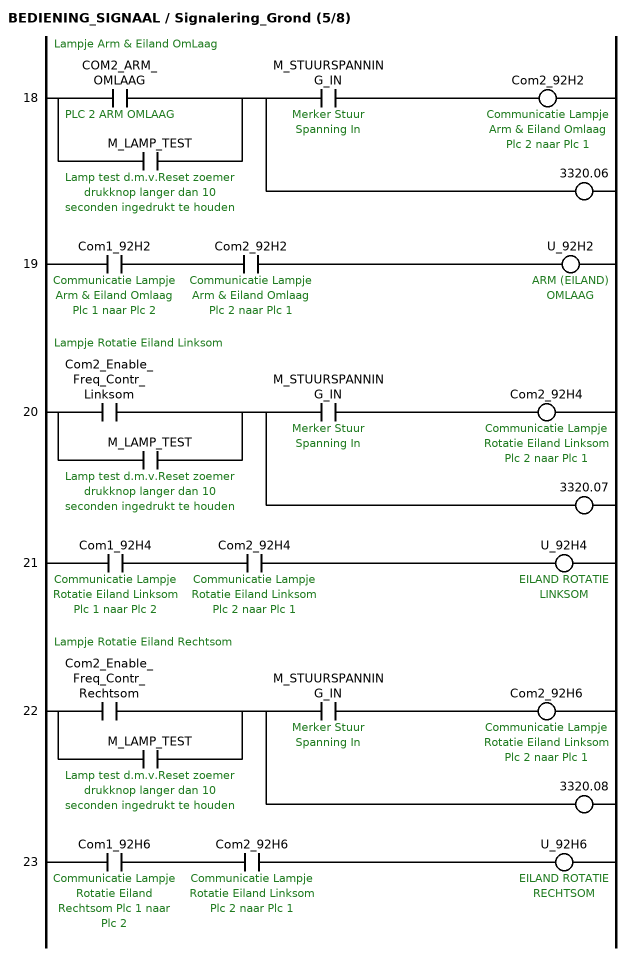
; [picture p301: BEDIENING_SIGNAAL / Signalering_Grond, rungs 18-23]
; rung 18: Lampje Arm & Eiland OmLaag
LD COM2_ARM_OMLAAG  ; PLC 2 ARM OMLAAG
OR M_LAMP_TEST  ; Lamp test d.m.v.Reset zoemer drukknop langer dan 10 seconden ingedrukt te houden
OUT TR0
AND M_STUURSPANNING_IN  ; Merker Stuur Spanning In
OUT Com2_92H2  ; Communicatie Lampje Arm & Eiland Omlaag Plc 2 naar Plc 1
LD TR0
OUT 3320.06
; rung 19
LD Com1_92H2  ; Communicatie Lampje Arm & Eiland Omlaag Plc 1 naar Plc 2
AND Com2_92H2  ; Communicatie Lampje Arm & Eiland Omlaag Plc 2 naar Plc 1
OUT U_92H2  ; ARM (EILAND) OMLAAG
; rung 20: Lampje Rotatie Eiland Linksom
LD Com2_Enable_Freq_Contr_Linksom
OR M_LAMP_TEST  ; Lamp test d.m.v.Reset zoemer drukknop langer dan 10 seconden ingedrukt te houden
OUT TR0
AND M_STUURSPANNING_IN  ; Merker Stuur Spanning In
OUT Com2_92H4  ; Communicatie Lampje Rotatie Eiland Linksom Plc 2 naar Plc 1
LD TR0
OUT 3320.07
; rung 21
LD Com1_92H4  ; Communicatie Lampje Rotatie Eiland Linksom Plc 1 naar Plc 2
AND Com2_92H4  ; Communicatie Lampje Rotatie Eiland Linksom Plc 2 naar Plc 1
OUT U_92H4  ; EILAND ROTATIE LINKSOM
; rung 22: Lampje Rotatie Eiland Rechtsom
LD Com2_Enable_Freq_Contr_Rechtsom
OR M_LAMP_TEST  ; Lamp test d.m.v.Reset zoemer drukknop langer dan 10 seconden ingedrukt te houden
OUT TR0
AND M_STUURSPANNING_IN  ; Merker Stuur Spanning In
OUT Com2_92H6  ; Communicatie Lampje Rotatie Eiland Linksom Plc 2 naar Plc 1
LD TR0
OUT 3320.08
; rung 23
LD Com1_92H6  ; Communicatie Lampje Rotatie Eiland Rechtsom Plc 1 naar Plc 2
AND Com2_92H6  ; Communicatie Lampje Rotatie Eiland Linksom Plc 2 naar Plc 1
OUT U_92H6  ; EILAND ROTATIE RECHTSOM

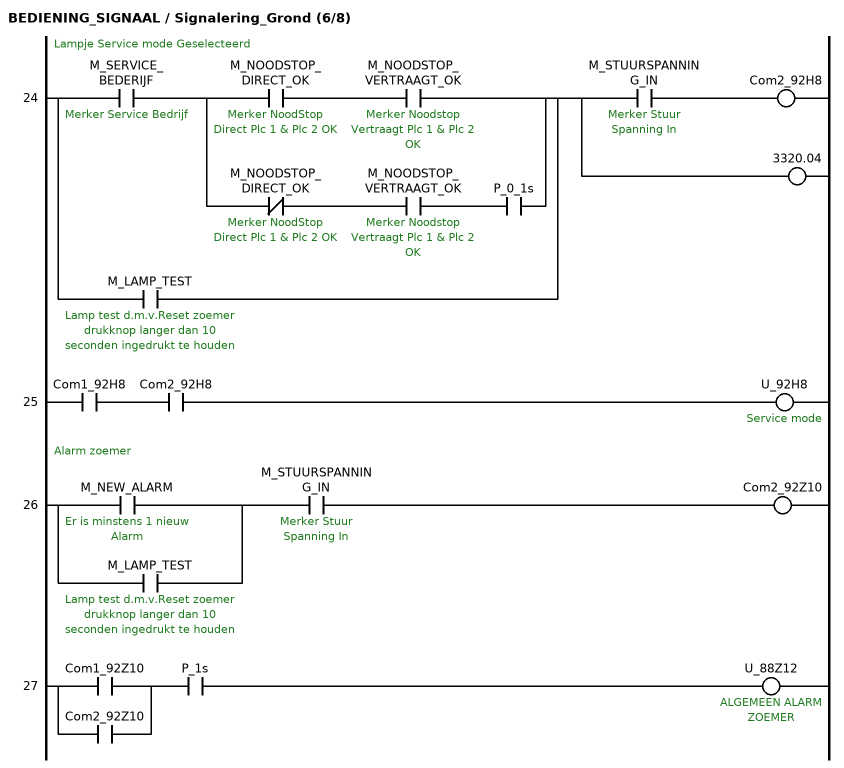
; rung 24: Lampje Service mode Geselecteerd
LD M_SERVICE_BEDERIJF  ; Merker Service Bedrijf
LD M_NOODSTOP_DIRECT_OK  ; Merker NoodStop Direct Plc 1 & Plc 2 OK
AND M_NOODSTOP_VERTRAAGT_OK  ; Merker Noodstop Vertraagt Plc 1 & Plc 2 OK
LDNOT M_NOODSTOP_DIRECT_OK  ; Merker NoodStop Direct Plc 1 & Plc 2 OK
AND M_NOODSTOP_VERTRAAGT_OK  ; Merker Noodstop Vertraagt Plc 1 & Plc 2 OK
AND P_0_1s
ORLD
ANDLD
OR M_LAMP_TEST  ; Lamp test d.m.v.Reset zoemer drukknop langer dan 10 seconden ingedrukt te houden
OUT TR0
AND M_STUURSPANNING_IN  ; Merker Stuur Spanning In
OUT Com2_92H8
LD TR0
OUT 3320.04
; rung 25
LD Com1_92H8
AND Com2_92H8
OUT U_92H8  ; Service mode
; rung 26: Alarm zoemer
LD M_NEW_ALARM  ; Er is minstens 1 nieuw Alarm
OR M_LAMP_TEST  ; Lamp test d.m.v.Reset zoemer drukknop langer dan 10 seconden ingedrukt te houden
AND M_STUURSPANNING_IN  ; Merker Stuur Spanning In
OUT Com2_92Z10
; rung 27
LD Com1_92Z10
OR Com2_92Z10
AND P_1s
OUT U_88Z12  ; ALGEMEEN ALARM ZOEMER

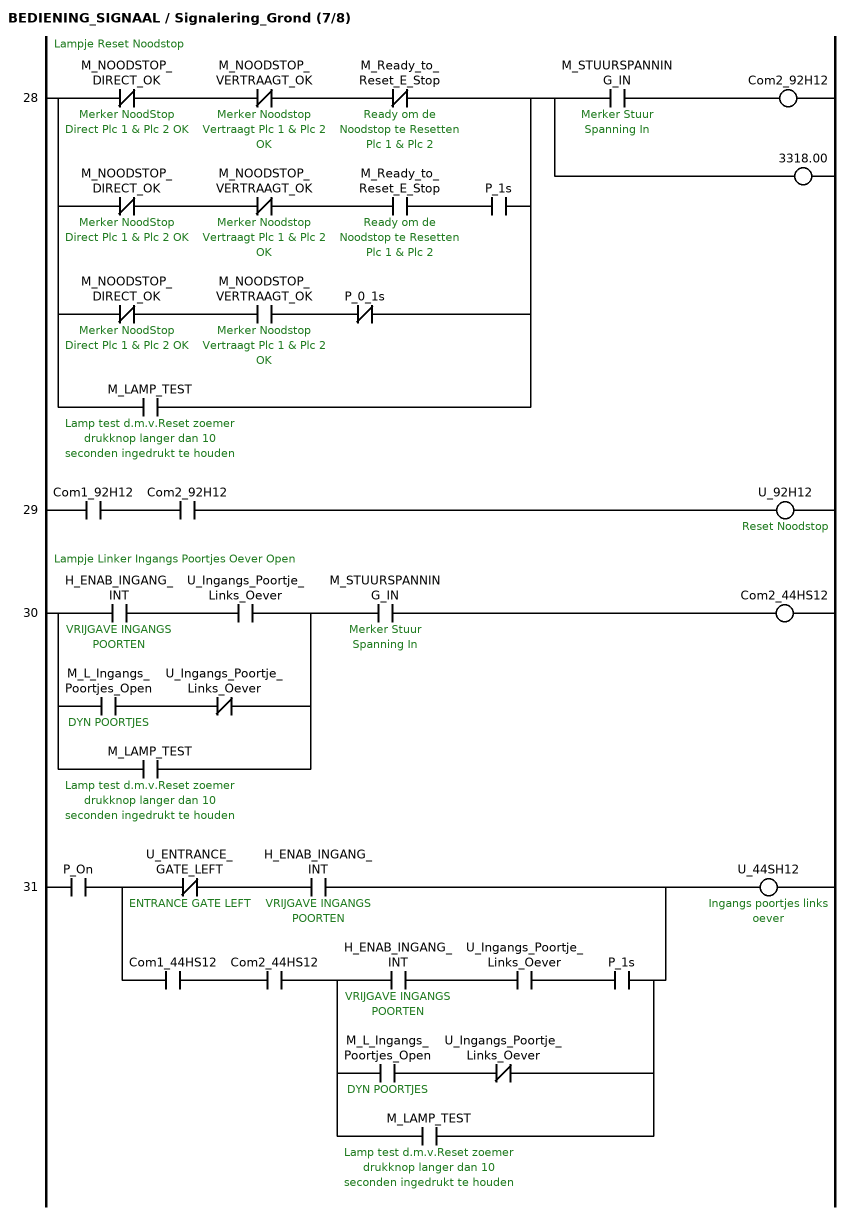
; rung 28: Lampje Reset Noodstop
LDNOT M_NOODSTOP_DIRECT_OK  ; Merker NoodStop Direct Plc 1 & Plc 2 OK
ANDNOT M_NOODSTOP_VERTRAAGT_OK  ; Merker Noodstop Vertraagt Plc 1 & Plc 2 OK
ANDNOT M_Ready_to_Reset_E_Stop  ; Ready om de Noodstop te Resetten Plc 1 & Plc 2
LDNOT M_NOODSTOP_DIRECT_OK  ; Merker NoodStop Direct Plc 1 & Plc 2 OK
ANDNOT M_NOODSTOP_VERTRAAGT_OK  ; Merker Noodstop Vertraagt Plc 1 & Plc 2 OK
AND M_Ready_to_Reset_E_Stop  ; Ready om de Noodstop te Resetten Plc 1 & Plc 2
AND P_1s
ORLD
LDNOT M_NOODSTOP_DIRECT_OK  ; Merker NoodStop Direct Plc 1 & Plc 2 OK
AND M_NOODSTOP_VERTRAAGT_OK  ; Merker Noodstop Vertraagt Plc 1 & Plc 2 OK
ANDNOT P_0_1s
ORLD
OR M_LAMP_TEST  ; Lamp test d.m.v.Reset zoemer drukknop langer dan 10 seconden ingedrukt te houden
OUT TR0
AND M_STUURSPANNING_IN  ; Merker Stuur Spanning In
OUT Com2_92H12
LD TR0
OUT 3318.00
; rung 29
LD Com1_92H12
AND Com2_92H12
OUT U_92H12  ; Reset Noodstop
; rung 30: Lampje Linker Ingangs Poortjes Oever Open
LD H_ENAB_INGANG_INT  ; VRIJGAVE INGANGS POORTEN
AND U_Ingangs_Poortje_Links_Oever
LD M_L_Ingangs_Poortjes_Open  ; DYN POORTJES
ANDNOT U_Ingangs_Poortje_Links_Oever
ORLD
OR M_LAMP_TEST  ; Lamp test d.m.v.Reset zoemer drukknop langer dan 10 seconden ingedrukt te houden
AND M_STUURSPANNING_IN  ; Merker Stuur Spanning In
OUT Com2_44HS12
; rung 31
LD P_On
LDNOT U_ENTRANCE_GATE_LEFT  ; ENTRANCE GATE LEFT
AND H_ENAB_INGANG_INT  ; VRIJGAVE INGANGS POORTEN
LD Com1_44HS12
AND Com2_44HS12
LD H_ENAB_INGANG_INT  ; VRIJGAVE INGANGS POORTEN
AND U_Ingangs_Poortje_Links_Oever
AND P_1s
LD M_L_Ingangs_Poortjes_Open  ; DYN POORTJES
ANDNOT U_Ingangs_Poortje_Links_Oever
ORLD
OR M_LAMP_TEST  ; Lamp test d.m.v.Reset zoemer drukknop langer dan 10 seconden ingedrukt te houden
ANDLD
ORLD
ANDLD
OUT U_44SH12  ; Ingangs poortjes links oever

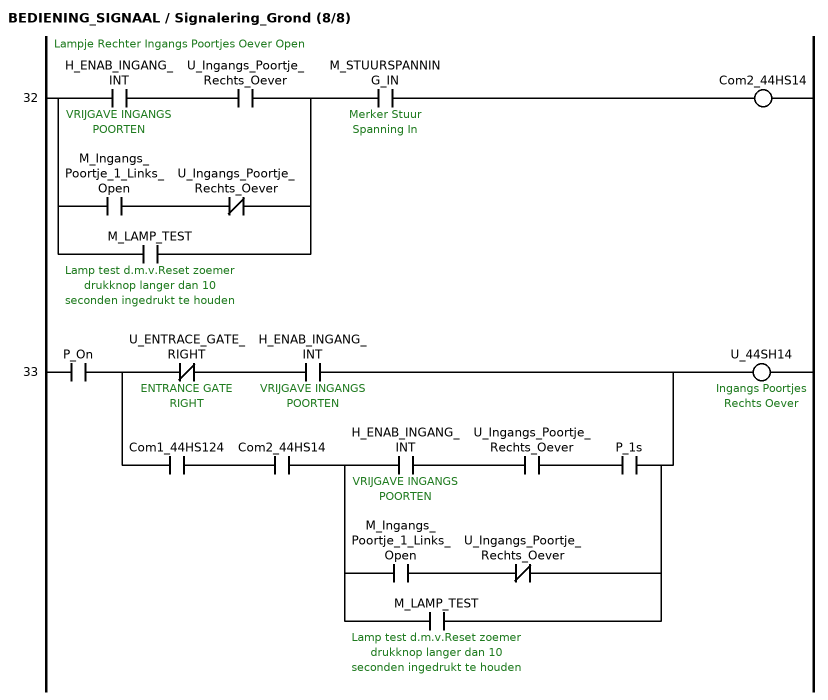
; rung 32: Lampje Rechter Ingangs Poortjes Oever Open
LD H_ENAB_INGANG_INT  ; VRIJGAVE INGANGS POORTEN
AND U_Ingangs_Poortje_Rechts_Oever
LD M_Ingangs_Poortje_1_Links_Open
ANDNOT U_Ingangs_Poortje_Rechts_Oever
ORLD
OR M_LAMP_TEST  ; Lamp test d.m.v.Reset zoemer drukknop langer dan 10 seconden ingedrukt te houden
AND M_STUURSPANNING_IN  ; Merker Stuur Spanning In
OUT Com2_44HS14
; rung 33
LD P_On
LDNOT U_ENTRACE_GATE_RIGHT  ; ENTRANCE GATE RIGHT
AND H_ENAB_INGANG_INT  ; VRIJGAVE INGANGS POORTEN
LD Com1_44HS124
AND Com2_44HS14
LD H_ENAB_INGANG_INT  ; VRIJGAVE INGANGS POORTEN
AND U_Ingangs_Poortje_Rechts_Oever
AND P_1s
LD M_Ingangs_Poortje_1_Links_Open
ANDNOT U_Ingangs_Poortje_Rechts_Oever
ORLD
OR M_LAMP_TEST  ; Lamp test d.m.v.Reset zoemer drukknop langer dan 10 seconden ingedrukt te houden
ANDLD
ORLD
ANDLD
OUT U_44SH14  ; Ingangs Poortjes Rechts Oever

### Section Bediening_Eiland

### Section Signalering_Eiland

### Section Bediening_Display_Eiland

### Section Signalering_Display_Eiland

### Section Einde_Bediening_Signalering
; rung 0
END(001)

## Program HOOFD_BESTURING (cyclic task 2)

### Section Automatische_Afloop_In_Uitgangs_Poortjes

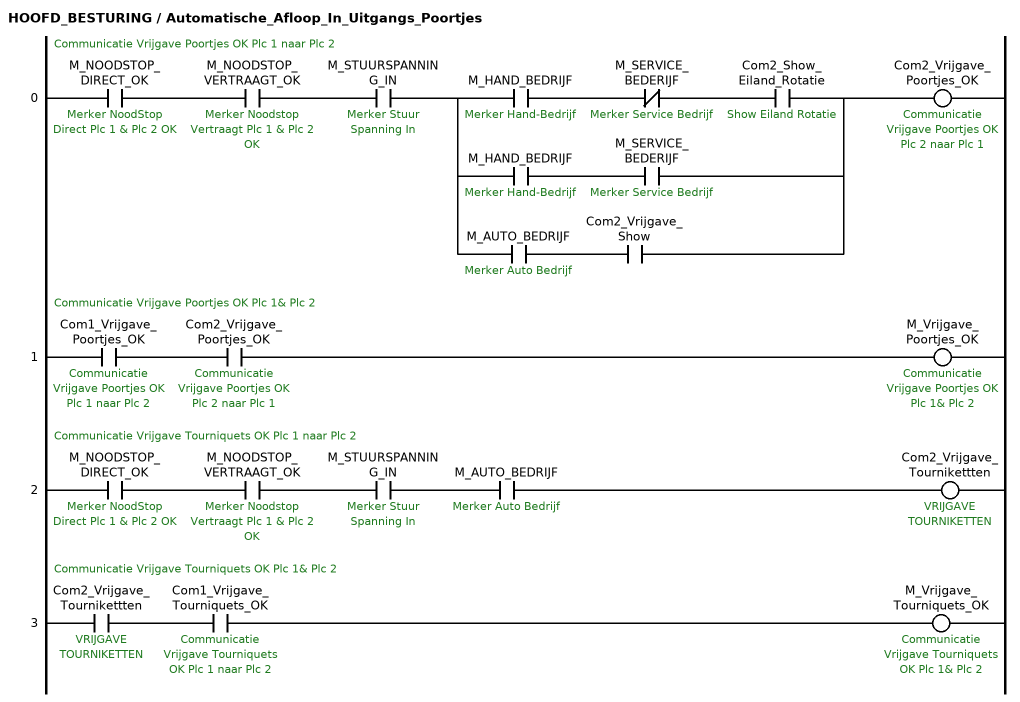
; rung 0: Communicatie Vrijgave Poortjes OK Plc 1 naar Plc 2
LD M_NOODSTOP_DIRECT_OK  ; Merker NoodStop Direct Plc 1 & Plc 2 OK
AND M_NOODSTOP_VERTRAAGT_OK  ; Merker Noodstop Vertraagt Plc 1 & Plc 2 OK
AND M_STUURSPANNING_IN  ; Merker Stuur Spanning In
LD M_HAND_BEDRIJF  ; Merker Hand-Bedrijf
ANDNOT M_SERVICE_BEDERIJF  ; Merker Service Bedrijf
AND Com2_Show_Eiland_Rotatie  ; Show Eiland Rotatie
LD M_HAND_BEDRIJF  ; Merker Hand-Bedrijf
AND M_SERVICE_BEDERIJF  ; Merker Service Bedrijf
ORLD
LD M_AUTO_BEDRIJF  ; Merker Auto Bedrijf
AND Com2_Vrijgave_Show
ORLD
ANDLD
OUT Com2_Vrijgave_Poortjes_OK  ; Communicatie Vrijgave Poortjes OK Plc 2 naar Plc 1
; rung 1: Communicatie Vrijgave Poortjes OK Plc 1& Plc 2
LD Com1_Vrijgave_Poortjes_OK  ; Communicatie Vrijgave Poortjes OK Plc 1 naar Plc 2
AND Com2_Vrijgave_Poortjes_OK  ; Communicatie Vrijgave Poortjes OK Plc 2 naar Plc 1
OUT M_Vrijgave_Poortjes_OK  ; Communicatie Vrijgave Poortjes OK Plc 1& Plc 2
; rung 2: Communicatie Vrijgave Tourniquets OK Plc 1 naar Plc 2
LD M_NOODSTOP_DIRECT_OK  ; Merker NoodStop Direct Plc 1 & Plc 2 OK
AND M_NOODSTOP_VERTRAAGT_OK  ; Merker Noodstop Vertraagt Plc 1 & Plc 2 OK
AND M_STUURSPANNING_IN  ; Merker Stuur Spanning In
AND M_AUTO_BEDRIJF  ; Merker Auto Bedrijf
OUT Com2_Vrijgave_Tournikettten  ; VRIJGAVE TOURNIKETTEN
; rung 3: Communicatie Vrijgave Tourniquets OK Plc 1& Plc 2
LD Com2_Vrijgave_Tournikettten  ; VRIJGAVE TOURNIKETTEN
AND Com1_Vrijgave_Tourniquets_OK  ; Communicatie Vrijgave Tourniquets OK Plc 1 naar Plc 2
OUT M_Vrijgave_Tourniquets_OK  ; Communicatie Vrijgave Tourniquets OK Plc 1& Plc 2

### Section Automatisch_Programma_Afloop

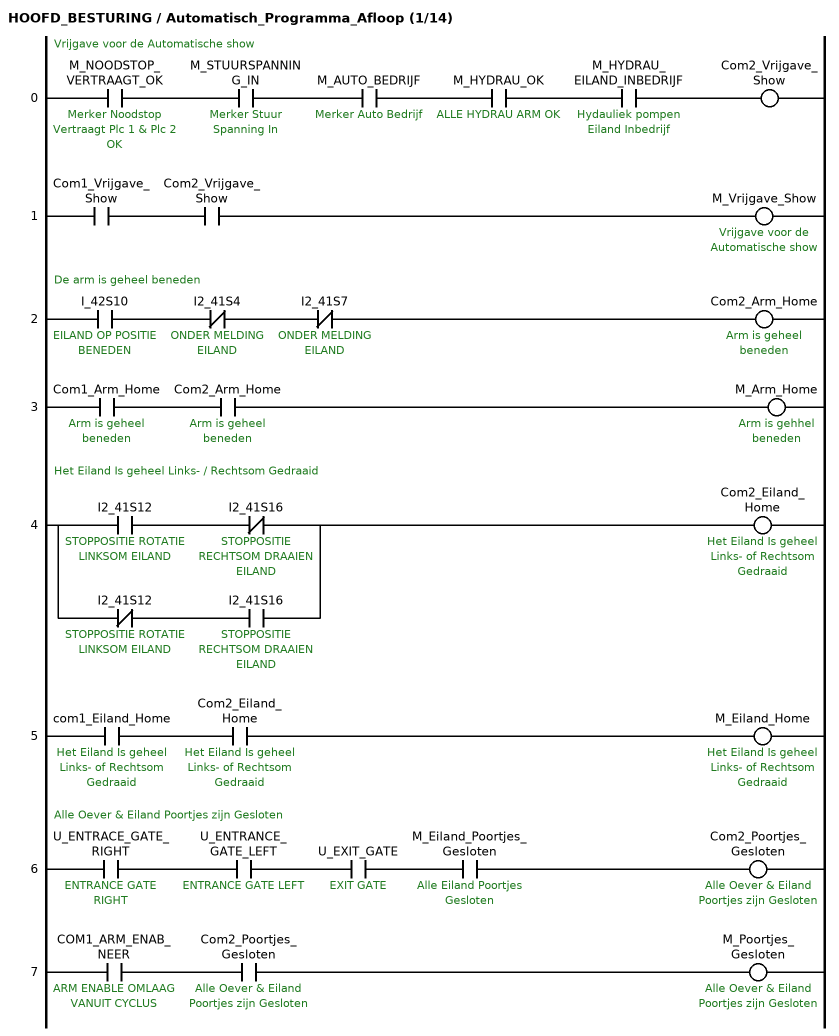
; rung 0: Vrijgave voor de Automatische show
LD M_NOODSTOP_VERTRAAGT_OK  ; Merker Noodstop Vertraagt Plc 1 & Plc 2 OK
AND M_STUURSPANNING_IN  ; Merker Stuur Spanning In
AND M_AUTO_BEDRIJF  ; Merker Auto Bedrijf
AND M_HYDRAU_OK  ; ALLE HYDRAU ARM OK
AND M_HYDRAU_EILAND_INBEDRIJF  ; Hydauliek pompen Eiland Inbedrijf
OUT Com2_Vrijgave_Show
; rung 1
LD Com1_Vrijgave_Show
AND Com2_Vrijgave_Show
OUT M_Vrijgave_Show  ; Vrijgave voor de Automatische show
; rung 2: De arm is geheel beneden
LD I_42S10  ; EILAND OP POSITIE BENEDEN
ANDNOT I2_41S4  ; ONDER MELDING EILAND
ANDNOT I2_41S7  ; ONDER MELDING EILAND
OUT Com2_Arm_Home  ; Arm is geheel beneden
; rung 3
LD Com1_Arm_Home  ; Arm is geheel beneden
AND Com2_Arm_Home  ; Arm is geheel beneden
OUT M_Arm_Home  ; Arm is gehhel beneden
; rung 4: Het Eiland Is geheel Links- / Rechtsom Gedraaid
LD I2_41S12  ; STOPPOSITIE ROTATIE LINKSOM EILAND
ANDNOT I2_41S16  ; STOPPOSITIE RECHTSOM DRAAIEN EILAND
LDNOT I2_41S12  ; STOPPOSITIE ROTATIE LINKSOM EILAND
AND I2_41S16  ; STOPPOSITIE RECHTSOM DRAAIEN EILAND
ORLD
OUT Com2_Eiland_Home  ; Het Eiland Is geheel Links- of Rechtsom Gedraaid
; rung 5
LD com1_Eiland_Home  ; Het Eiland Is geheel Links- of Rechtsom Gedraaid
AND Com2_Eiland_Home  ; Het Eiland Is geheel Links- of Rechtsom Gedraaid
OUT M_Eiland_Home  ; Het Eiland Is geheel Links- of Rechtsom Gedraaid
; rung 6: Alle Oever & Eiland Poortjes zijn Gesloten
LD U_ENTRACE_GATE_RIGHT  ; ENTRANCE GATE RIGHT
AND U_ENTRANCE_GATE_LEFT  ; ENTRANCE GATE LEFT
AND U_EXIT_GATE  ; EXIT GATE
AND M_Eiland_Poortjes_Gesloten  ; Alle Eiland Poortjes Gesloten
OUT Com2_Poortjes_Gesloten  ; Alle Oever & Eiland Poortjes zijn Gesloten
; rung 7
LD COM1_ARM_ENAB_NEER  ; ARM ENABLE OMLAAG  VANUIT CYCLUS
AND Com2_Poortjes_Gesloten  ; Alle Oever & Eiland Poortjes zijn Gesloten
OUT M_Poortjes_Gesloten  ; Alle Oever & Eiland Poortjes zijn Gesloten

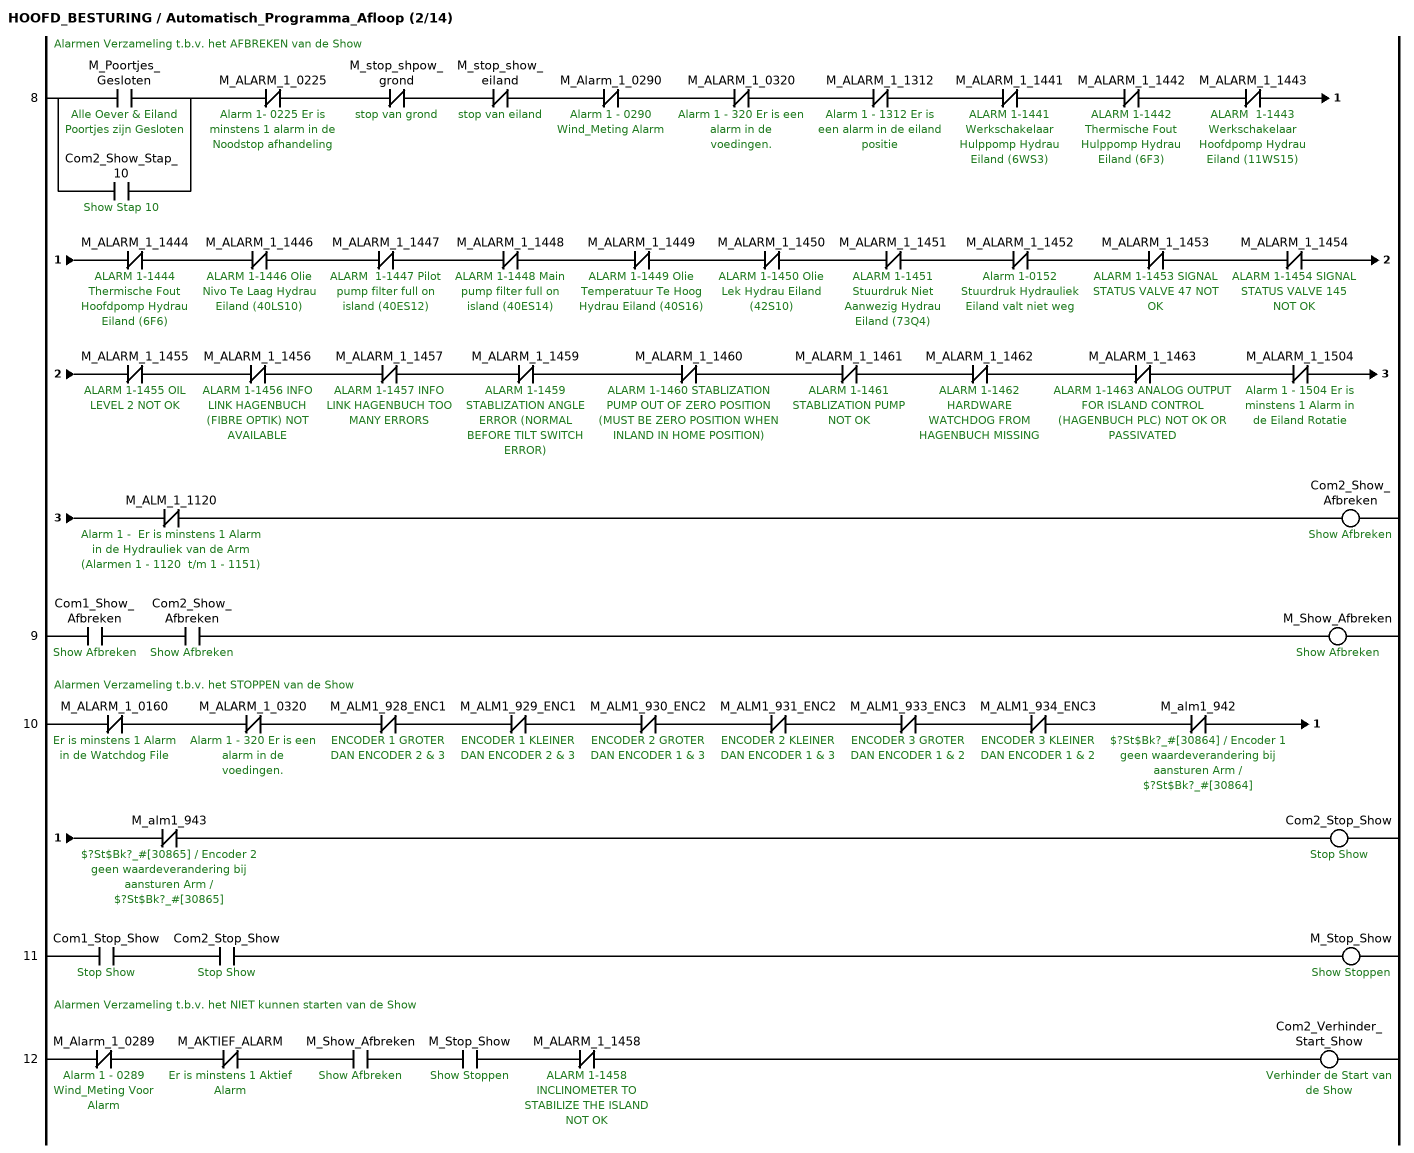
; rung 8: Alarmen Verzameling t.b.v. het AFBREKEN van de Show
LD M_Poortjes_Gesloten  ; Alle Oever & Eiland Poortjes zijn Gesloten
OR Com2_Show_Stap_10  ; Show Stap 10
ANDNOT M_ALARM_1_0225  ; Alarm 1- 0225 Er is minstens 1 alarm in de Noodstop afhandeling
ANDNOT M_stop_shpow_grond  ; stop van grond
ANDNOT M_stop_show_eiland  ; stop van eiland
ANDNOT M_Alarm_1_0290  ; Alarm 1 - 0290 Wind_Meting Alarm
ANDNOT M_ALARM_1_0320  ; Alarm 1 - 320 Er is een alarm in de voedingen.
ANDNOT M_ALARM_1_1312  ; Alarm 1 - 1312 Er is een alarm in de eiland positie
ANDNOT M_ALARM_1_1441  ; ALARM 1-1441 Werkschakelaar Hulppomp Hydrau Eiland (6WS3)
ANDNOT M_ALARM_1_1442  ; ALARM 1-1442 Thermische Fout Hulppomp Hydrau Eiland (6F3)
ANDNOT M_ALARM_1_1443  ; ALARM  1-1443 Werkschakelaar Hoofdpomp Hydrau Eiland (11WS15)
ANDNOT M_ALARM_1_1444  ; ALARM 1-1444 Thermische Fout Hoofdpomp Hydrau Eiland (6F6)
ANDNOT M_ALARM_1_1446  ; ALARM 1-1446 Olie Nivo Te Laag Hydrau Eiland (40LS10)
ANDNOT M_ALARM_1_1447  ; ALARM  1-1447 Pilot pump filter full on island (40ES12)
ANDNOT M_ALARM_1_1448  ; ALARM 1-1448 Main pump filter full on island (40ES14)
ANDNOT M_ALARM_1_1449  ; ALARM 1-1449 Olie Temperatuur Te Hoog Hydrau Eiland (40S16)
ANDNOT M_ALARM_1_1450  ; ALARM 1-1450 Olie Lek Hydrau Eiland (42S10)
ANDNOT M_ALARM_1_1451  ; ALARM 1-1451 Stuurdruk Niet Aanwezig Hydrau Eiland (73Q4)
ANDNOT M_ALARM_1_1452  ; Alarm 1-0152 Stuurdruk Hydrauliek Eiland valt niet weg
ANDNOT M_ALARM_1_1453  ; ALARM 1-1453 SIGNAL STATUS VALVE 47 NOT OK
ANDNOT M_ALARM_1_1454  ; ALARM 1-1454 SIGNAL STATUS VALVE 145 NOT OK
ANDNOT M_ALARM_1_1455  ; ALARM 1-1455 OIL LEVEL 2 NOT OK
ANDNOT M_ALARM_1_1456  ; ALARM 1-1456 INFO LINK HAGENBUCH (FIBRE OPTIK) NOT AVAILABLE
ANDNOT M_ALARM_1_1457  ; ALARM 1-1457 INFO LINK HAGENBUCH TOO MANY ERRORS
ANDNOT M_ALARM_1_1459  ; ALARM 1-1459 STABLIZATION ANGLE ERROR (NORMAL BEFORE TILT SWITCH ERROR)
ANDNOT M_ALARM_1_1460  ; ALARM 1-1460 STABLIZATION PUMP OUT OF ZERO POSITION (MUST BE ZERO POSITION WHEN INLAND IN HOME POSITION)
ANDNOT M_ALARM_1_1461  ; ALARM 1-1461 STABLIZATION PUMP NOT OK
ANDNOT M_ALARM_1_1462  ; ALARM 1-1462 HARDWARE WATCHDOG FROM HAGENBUCH MISSING
ANDNOT M_ALARM_1_1463  ; ALARM 1-1463 ANALOG OUTPUT FOR ISLAND CONTROL (HAGENBUCH PLC) NOT OK OR PASSIVATED
ANDNOT M_ALARM_1_1504  ; Alarm 1 - 1504 Er is minstens 1 Alarm in de Eiland Rotatie
ANDNOT M_ALM_1_1120  ; Alarm 1 -  Er is minstens 1 Alarm in de Hydrauliek van de Arm  (Alarmen 1 - 1120  t/m 1 - 1151)
OUT Com2_Show_Afbreken  ; Show Afbreken
; rung 9
LD Com1_Show_Afbreken  ; Show Afbreken
AND Com2_Show_Afbreken  ; Show Afbreken
OUT M_Show_Afbreken  ; Show Afbreken
; rung 10: Alarmen Verzameling t.b.v. het STOPPEN van de Show
LDNOT M_ALARM_1_0160  ; Er is minstens 1 Alarm in de Watchdog File
ANDNOT M_ALARM_1_0320  ; Alarm 1 - 320 Er is een alarm in de voedingen.
ANDNOT M_ALM1_928_ENC1  ; ENCODER 1 GROTER DAN ENCODER 2 & 3
ANDNOT M_ALM1_929_ENC1  ; ENCODER 1 KLEINER DAN ENCODER 2 & 3
ANDNOT M_ALM1_930_ENC2  ; ENCODER 2 GROTER DAN ENCODER 1 & 3
ANDNOT M_ALM1_931_ENC2  ; ENCODER 2 KLEINER DAN ENCODER 1 & 3
ANDNOT M_ALM1_933_ENC3  ; ENCODER 3 GROTER DAN ENCODER 1 & 2
ANDNOT M_ALM1_934_ENC3  ; ENCODER 3 KLEINER DAN ENCODER 1 & 2
ANDNOT M_alm1_942  ; $?St$Bk?_#[30864] / Encoder 1 geen waardeverandering bij aansturen Arm / $?St$Bk?_#[30864]
ANDNOT M_alm1_943  ; $?St$Bk?_#[30865] / Encoder 2 geen waardeverandering bij aansturen Arm / $?St$Bk?_#[30865]
OUT Com2_Stop_Show  ; Stop Show
; rung 11
LD Com1_Stop_Show  ; Stop Show
AND Com2_Stop_Show  ; Stop Show
OUT M_Stop_Show  ; Show Stoppen
; rung 12: Alarmen Verzameling t.b.v. het NIET kunnen starten van de Show
LDNOT M_Alarm_1_0289  ; Alarm 1 - 0289 Wind_Meting Voor Alarm
ANDNOT M_AKTIEF_ALARM  ; Er is minstens 1 Aktief Alarm
AND M_Show_Afbreken  ; Show Afbreken
AND M_Stop_Show  ; Show Stoppen
ANDNOT M_ALARM_1_1458  ; ALARM 1-1458 INCLINOMETER TO STABILIZE THE ISLAND NOT OK
OUT Com2_Verhinder_Start_Show  ; Verhinder de Start van de Show

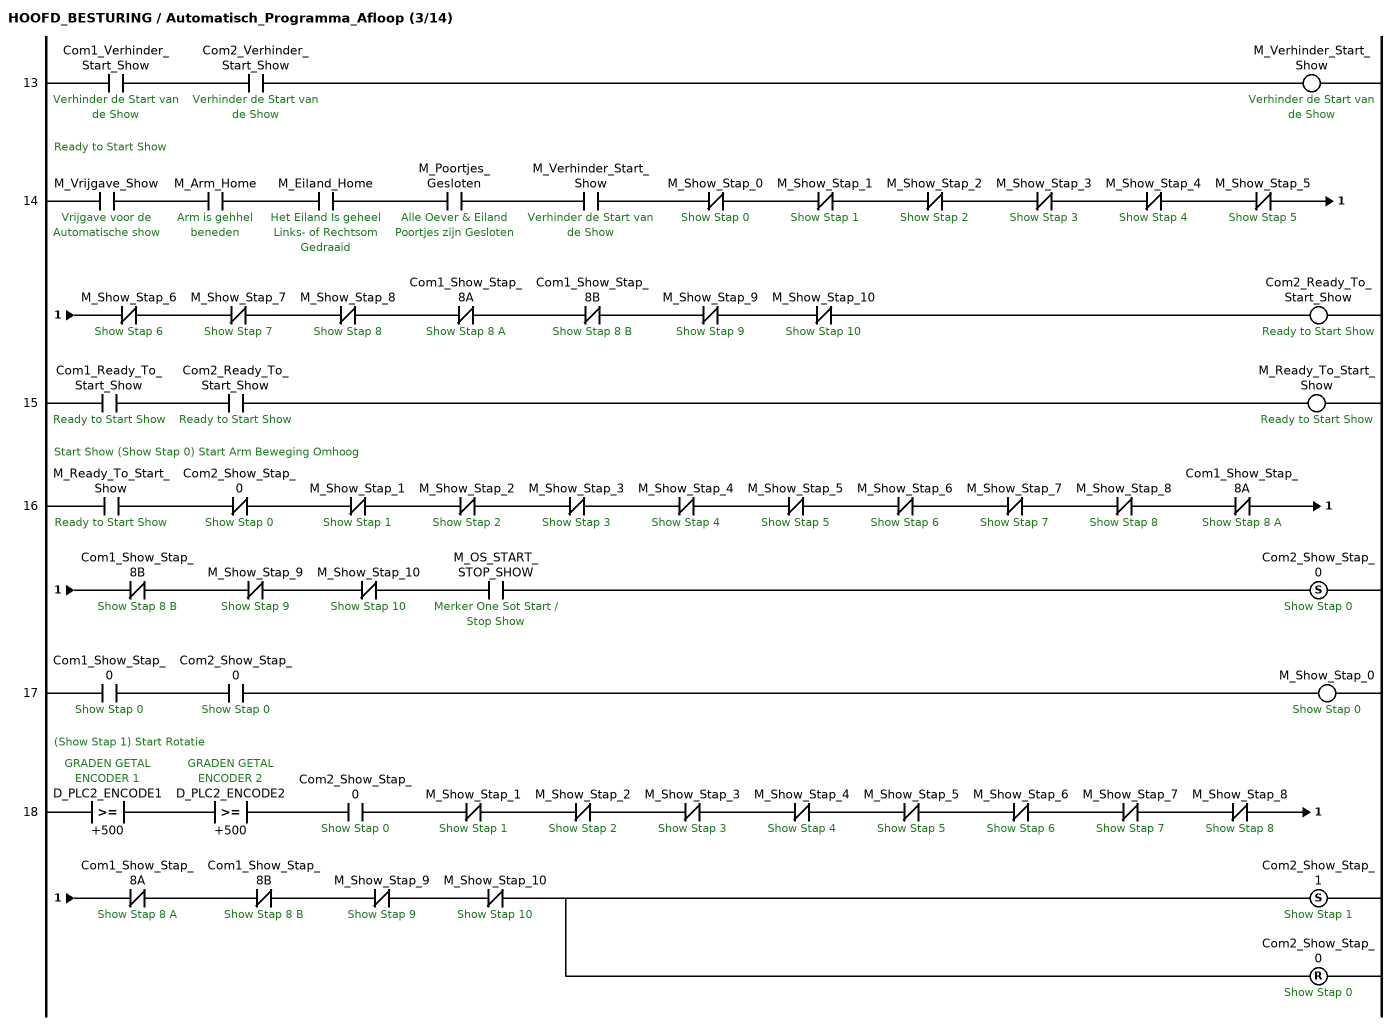
; rung 13
LD Com1_Verhinder_Start_Show  ; Verhinder de Start van de Show
AND Com2_Verhinder_Start_Show  ; Verhinder de Start van de Show
OUT M_Verhinder_Start_Show  ; Verhinder de Start van de Show
; rung 14: Ready to Start Show
LD M_Vrijgave_Show  ; Vrijgave voor de Automatische show
AND M_Arm_Home  ; Arm is gehhel beneden
AND M_Eiland_Home  ; Het Eiland Is geheel Links- of Rechtsom Gedraaid
AND M_Poortjes_Gesloten  ; Alle Oever & Eiland Poortjes zijn Gesloten
AND M_Verhinder_Start_Show  ; Verhinder de Start van de Show
ANDNOT M_Show_Stap_0  ; Show Stap 0
ANDNOT M_Show_Stap_1  ; Show Stap 1
ANDNOT M_Show_Stap_2  ; Show Stap 2
ANDNOT M_Show_Stap_3  ; Show Stap 3
ANDNOT M_Show_Stap_4  ; Show Stap 4
ANDNOT M_Show_Stap_5  ; Show Stap 5
ANDNOT M_Show_Stap_6  ; Show Stap 6
ANDNOT M_Show_Stap_7  ; Show Stap 7
ANDNOT M_Show_Stap_8  ; Show Stap 8
ANDNOT Com1_Show_Stap_8A  ; Show Stap 8 A
ANDNOT Com1_Show_Stap_8B  ; Show Stap 8 B
ANDNOT M_Show_Stap_9  ; Show Stap 9
ANDNOT M_Show_Stap_10  ; Show Stap 10
OUT Com2_Ready_To_Start_Show  ; Ready to Start Show
; rung 15
LD Com1_Ready_To_Start_Show  ; Ready to Start Show
AND Com2_Ready_To_Start_Show  ; Ready to Start Show
OUT M_Ready_To_Start_Show  ; Ready to Start Show
; rung 16: Start Show (Show Stap 0) Start Arm Beweging Omhoog
LD M_Ready_To_Start_Show  ; Ready to Start Show
ANDNOT Com2_Show_Stap_0  ; Show Stap 0
ANDNOT M_Show_Stap_1  ; Show Stap 1
ANDNOT M_Show_Stap_2  ; Show Stap 2
ANDNOT M_Show_Stap_3  ; Show Stap 3
ANDNOT M_Show_Stap_4  ; Show Stap 4
ANDNOT M_Show_Stap_5  ; Show Stap 5
ANDNOT M_Show_Stap_6  ; Show Stap 6
ANDNOT M_Show_Stap_7  ; Show Stap 7
ANDNOT M_Show_Stap_8  ; Show Stap 8
ANDNOT Com1_Show_Stap_8A  ; Show Stap 8 A
ANDNOT Com1_Show_Stap_8B  ; Show Stap 8 B
ANDNOT M_Show_Stap_9  ; Show Stap 9
ANDNOT M_Show_Stap_10  ; Show Stap 10
AND M_OS_START_STOP_SHOW  ; Merker One Sot Start / Stop Show
SET Com2_Show_Stap_0  ; Show Stap 0
; rung 17
LD Com1_Show_Stap_0  ; Show Stap 0
AND Com2_Show_Stap_0  ; Show Stap 0
OUT M_Show_Stap_0  ; Show Stap 0
; rung 18: (Show Stap 1) Start Rotatie
LD>=S(327) D_PLC2_ENCODE1 +500  ; GRADEN GETAL ENCODER 1
AND>=S(327) D_PLC2_ENCODE2 +500  ; GRADEN GETAL ENCODER 2
AND Com2_Show_Stap_0  ; Show Stap 0
ANDNOT M_Show_Stap_1  ; Show Stap 1
ANDNOT M_Show_Stap_2  ; Show Stap 2
ANDNOT M_Show_Stap_3  ; Show Stap 3
ANDNOT M_Show_Stap_4  ; Show Stap 4
ANDNOT M_Show_Stap_5  ; Show Stap 5
ANDNOT M_Show_Stap_6  ; Show Stap 6
ANDNOT M_Show_Stap_7  ; Show Stap 7
ANDNOT M_Show_Stap_8  ; Show Stap 8
ANDNOT Com1_Show_Stap_8A  ; Show Stap 8 A
ANDNOT Com1_Show_Stap_8B  ; Show Stap 8 B
ANDNOT M_Show_Stap_9  ; Show Stap 9
ANDNOT M_Show_Stap_10  ; Show Stap 10
SET Com2_Show_Stap_1  ; Show Stap 1
RSET Com2_Show_Stap_0  ; Show Stap 0

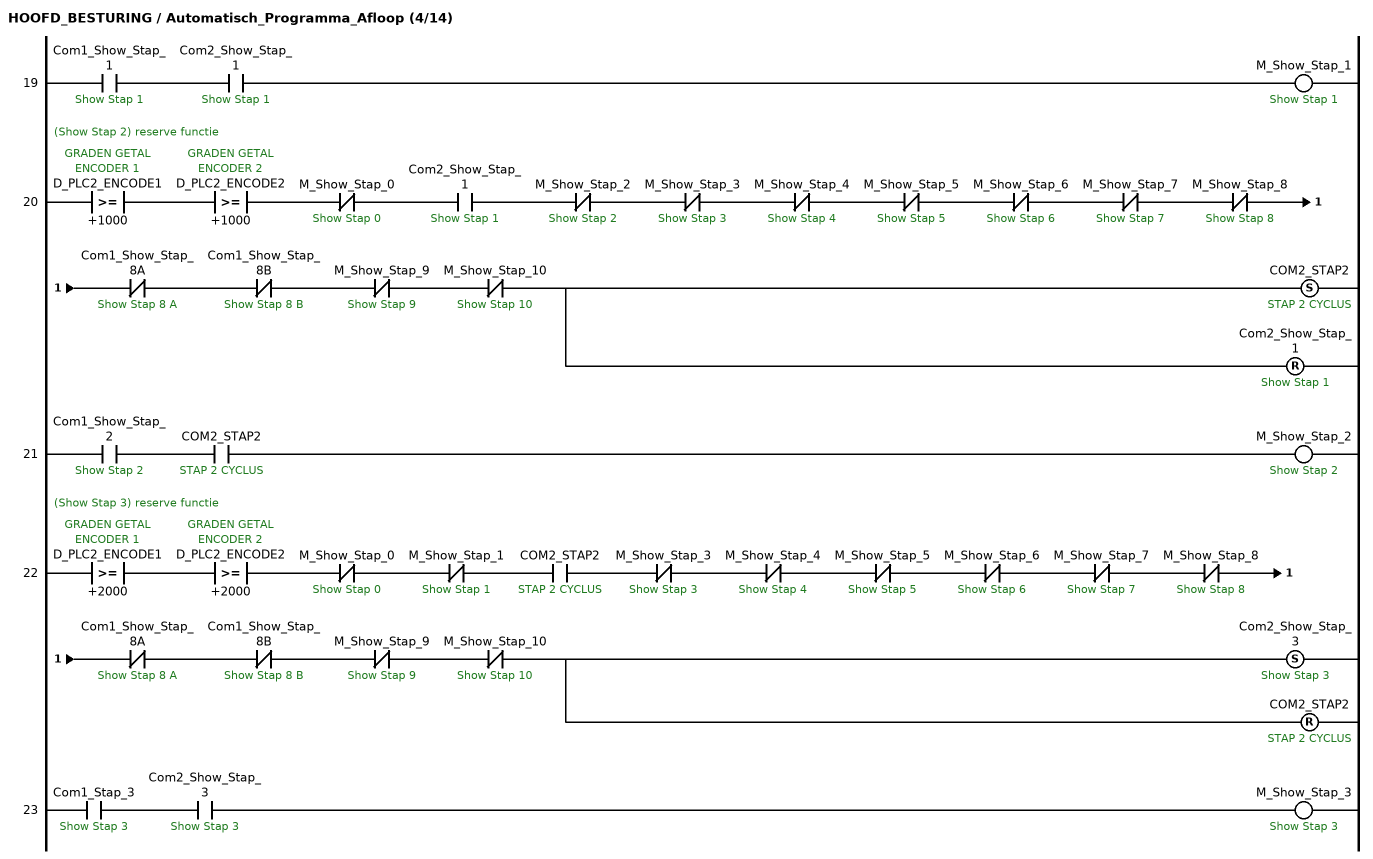
; rung 19
LD Com1_Show_Stap_1  ; Show Stap 1
AND Com2_Show_Stap_1  ; Show Stap 1
OUT M_Show_Stap_1  ; Show Stap 1
; rung 20: (Show Stap 2) reserve functie
LD>=S(327) D_PLC2_ENCODE1 +1000  ; GRADEN GETAL ENCODER 1
AND>=S(327) D_PLC2_ENCODE2 +1000  ; GRADEN GETAL ENCODER 2
ANDNOT M_Show_Stap_0  ; Show Stap 0
AND Com2_Show_Stap_1  ; Show Stap 1
ANDNOT M_Show_Stap_2  ; Show Stap 2
ANDNOT M_Show_Stap_3  ; Show Stap 3
ANDNOT M_Show_Stap_4  ; Show Stap 4
ANDNOT M_Show_Stap_5  ; Show Stap 5
ANDNOT M_Show_Stap_6  ; Show Stap 6
ANDNOT M_Show_Stap_7  ; Show Stap 7
ANDNOT M_Show_Stap_8  ; Show Stap 8
ANDNOT Com1_Show_Stap_8A  ; Show Stap 8 A
ANDNOT Com1_Show_Stap_8B  ; Show Stap 8 B
ANDNOT M_Show_Stap_9  ; Show Stap 9
ANDNOT M_Show_Stap_10  ; Show Stap 10
SET COM2_STAP2  ; STAP 2 CYCLUS
RSET Com2_Show_Stap_1  ; Show Stap 1
; rung 21
LD Com1_Show_Stap_2  ; Show Stap 2
AND COM2_STAP2  ; STAP 2 CYCLUS
OUT M_Show_Stap_2  ; Show Stap 2
; rung 22: (Show Stap 3) reserve functie
LD>=S(327) D_PLC2_ENCODE1 +2000  ; GRADEN GETAL ENCODER 1
AND>=S(327) D_PLC2_ENCODE2 +2000  ; GRADEN GETAL ENCODER 2
ANDNOT M_Show_Stap_0  ; Show Stap 0
ANDNOT M_Show_Stap_1  ; Show Stap 1
AND COM2_STAP2  ; STAP 2 CYCLUS
ANDNOT M_Show_Stap_3  ; Show Stap 3
ANDNOT M_Show_Stap_4  ; Show Stap 4
ANDNOT M_Show_Stap_5  ; Show Stap 5
ANDNOT M_Show_Stap_6  ; Show Stap 6
ANDNOT M_Show_Stap_7  ; Show Stap 7
ANDNOT M_Show_Stap_8  ; Show Stap 8
ANDNOT Com1_Show_Stap_8A  ; Show Stap 8 A
ANDNOT Com1_Show_Stap_8B  ; Show Stap 8 B
ANDNOT M_Show_Stap_9  ; Show Stap 9
ANDNOT M_Show_Stap_10  ; Show Stap 10
SET Com2_Show_Stap_3  ; Show Stap 3
RSET COM2_STAP2  ; STAP 2 CYCLUS
; rung 23
LD Com1_Stap_3  ; Show Stap 3
AND Com2_Show_Stap_3  ; Show Stap 3
OUT M_Show_Stap_3  ; Show Stap 3

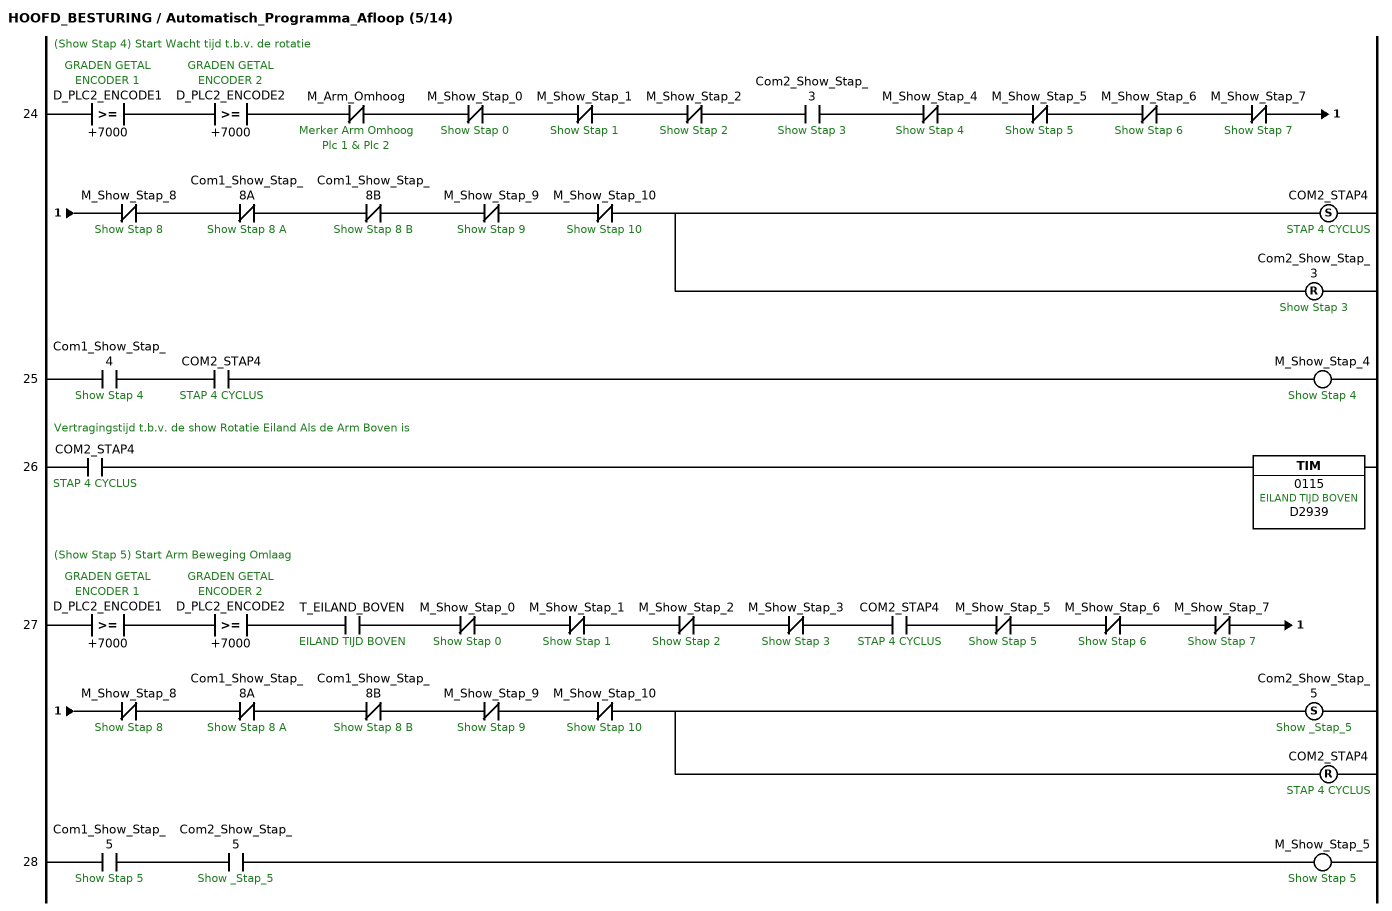
; rung 24: (Show Stap 4) Start Wacht tijd t.b.v. de rotatie
LD>=S(327) D_PLC2_ENCODE1 +7000  ; GRADEN GETAL ENCODER 1
AND>=S(327) D_PLC2_ENCODE2 +7000  ; GRADEN GETAL ENCODER 2
ANDNOT M_Arm_Omhoog  ; Merker Arm Omhoog Plc 1 & Plc 2
ANDNOT M_Show_Stap_0  ; Show Stap 0
ANDNOT M_Show_Stap_1  ; Show Stap 1
ANDNOT M_Show_Stap_2  ; Show Stap 2
AND Com2_Show_Stap_3  ; Show Stap 3
ANDNOT M_Show_Stap_4  ; Show Stap 4
ANDNOT M_Show_Stap_5  ; Show Stap 5
ANDNOT M_Show_Stap_6  ; Show Stap 6
ANDNOT M_Show_Stap_7  ; Show Stap 7
ANDNOT M_Show_Stap_8  ; Show Stap 8
ANDNOT Com1_Show_Stap_8A  ; Show Stap 8 A
ANDNOT Com1_Show_Stap_8B  ; Show Stap 8 B
ANDNOT M_Show_Stap_9  ; Show Stap 9
ANDNOT M_Show_Stap_10  ; Show Stap 10
SET COM2_STAP4  ; STAP 4 CYCLUS
RSET Com2_Show_Stap_3  ; Show Stap 3
; rung 25
LD Com1_Show_Stap_4  ; Show Stap 4
AND COM2_STAP4  ; STAP 4 CYCLUS
OUT M_Show_Stap_4  ; Show Stap 4
; rung 26: Vertragingstijd t.b.v. de show Rotatie Eiland Als de Arm Boven is
LD COM2_STAP4  ; STAP 4 CYCLUS
TIM 0115 D2939  ; EILAND TIJD BOVEN
; rung 27: (Show Stap 5) Start Arm Beweging Omlaag
LD>=S(327) D_PLC2_ENCODE1 +7000  ; GRADEN GETAL ENCODER 1
AND>=S(327) D_PLC2_ENCODE2 +7000  ; GRADEN GETAL ENCODER 2
AND T_EILAND_BOVEN  ; EILAND TIJD BOVEN
ANDNOT M_Show_Stap_0  ; Show Stap 0
ANDNOT M_Show_Stap_1  ; Show Stap 1
ANDNOT M_Show_Stap_2  ; Show Stap 2
ANDNOT M_Show_Stap_3  ; Show Stap 3
AND COM2_STAP4  ; STAP 4 CYCLUS
ANDNOT M_Show_Stap_5  ; Show Stap 5
ANDNOT M_Show_Stap_6  ; Show Stap 6
ANDNOT M_Show_Stap_7  ; Show Stap 7
ANDNOT M_Show_Stap_8  ; Show Stap 8
ANDNOT Com1_Show_Stap_8A  ; Show Stap 8 A
ANDNOT Com1_Show_Stap_8B  ; Show Stap 8 B
ANDNOT M_Show_Stap_9  ; Show Stap 9
ANDNOT M_Show_Stap_10  ; Show Stap 10
SET Com2_Show_Stap_5  ; Show _Stap_5
RSET COM2_STAP4  ; STAP 4 CYCLUS
; rung 28
LD Com1_Show_Stap_5  ; Show Stap 5
AND Com2_Show_Stap_5  ; Show _Stap_5
OUT M_Show_Stap_5  ; Show Stap 5

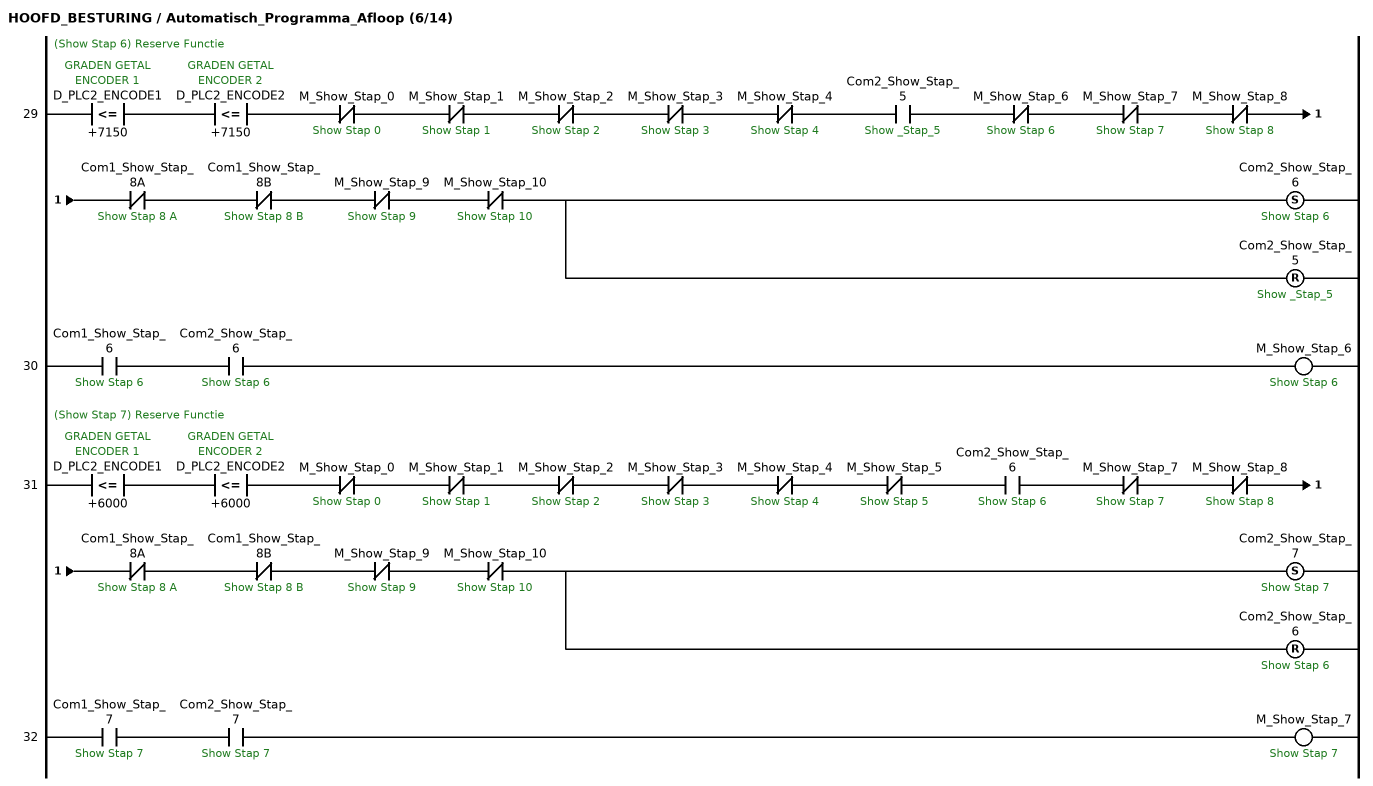
; rung 29: (Show Stap 6) Reserve Functie
LD<=S(317) D_PLC2_ENCODE1 +7150  ; GRADEN GETAL ENCODER 1
AND<=S(317) D_PLC2_ENCODE2 +7150  ; GRADEN GETAL ENCODER 2
ANDNOT M_Show_Stap_0  ; Show Stap 0
ANDNOT M_Show_Stap_1  ; Show Stap 1
ANDNOT M_Show_Stap_2  ; Show Stap 2
ANDNOT M_Show_Stap_3  ; Show Stap 3
ANDNOT M_Show_Stap_4  ; Show Stap 4
AND Com2_Show_Stap_5  ; Show _Stap_5
ANDNOT M_Show_Stap_6  ; Show Stap 6
ANDNOT M_Show_Stap_7  ; Show Stap 7
ANDNOT M_Show_Stap_8  ; Show Stap 8
ANDNOT Com1_Show_Stap_8A  ; Show Stap 8 A
ANDNOT Com1_Show_Stap_8B  ; Show Stap 8 B
ANDNOT M_Show_Stap_9  ; Show Stap 9
ANDNOT M_Show_Stap_10  ; Show Stap 10
SET Com2_Show_Stap_6  ; Show Stap 6
RSET Com2_Show_Stap_5  ; Show _Stap_5
; rung 30
LD Com1_Show_Stap_6  ; Show Stap 6
AND Com2_Show_Stap_6  ; Show Stap 6
OUT M_Show_Stap_6  ; Show Stap 6
; rung 31: (Show Stap 7) Reserve Functie
LD<=S(317) D_PLC2_ENCODE1 +6000  ; GRADEN GETAL ENCODER 1
AND<=S(317) D_PLC2_ENCODE2 +6000  ; GRADEN GETAL ENCODER 2
ANDNOT M_Show_Stap_0  ; Show Stap 0
ANDNOT M_Show_Stap_1  ; Show Stap 1
ANDNOT M_Show_Stap_2  ; Show Stap 2
ANDNOT M_Show_Stap_3  ; Show Stap 3
ANDNOT M_Show_Stap_4  ; Show Stap 4
ANDNOT M_Show_Stap_5  ; Show Stap 5
AND Com2_Show_Stap_6  ; Show Stap 6
ANDNOT M_Show_Stap_7  ; Show Stap 7
ANDNOT M_Show_Stap_8  ; Show Stap 8
ANDNOT Com1_Show_Stap_8A  ; Show Stap 8 A
ANDNOT Com1_Show_Stap_8B  ; Show Stap 8 B
ANDNOT M_Show_Stap_9  ; Show Stap 9
ANDNOT M_Show_Stap_10  ; Show Stap 10
SET Com2_Show_Stap_7  ; Show Stap 7
RSET Com2_Show_Stap_6  ; Show Stap 6
; rung 32
LD Com1_Show_Stap_7  ; Show Stap 7
AND Com2_Show_Stap_7  ; Show Stap 7
OUT M_Show_Stap_7  ; Show Stap 7

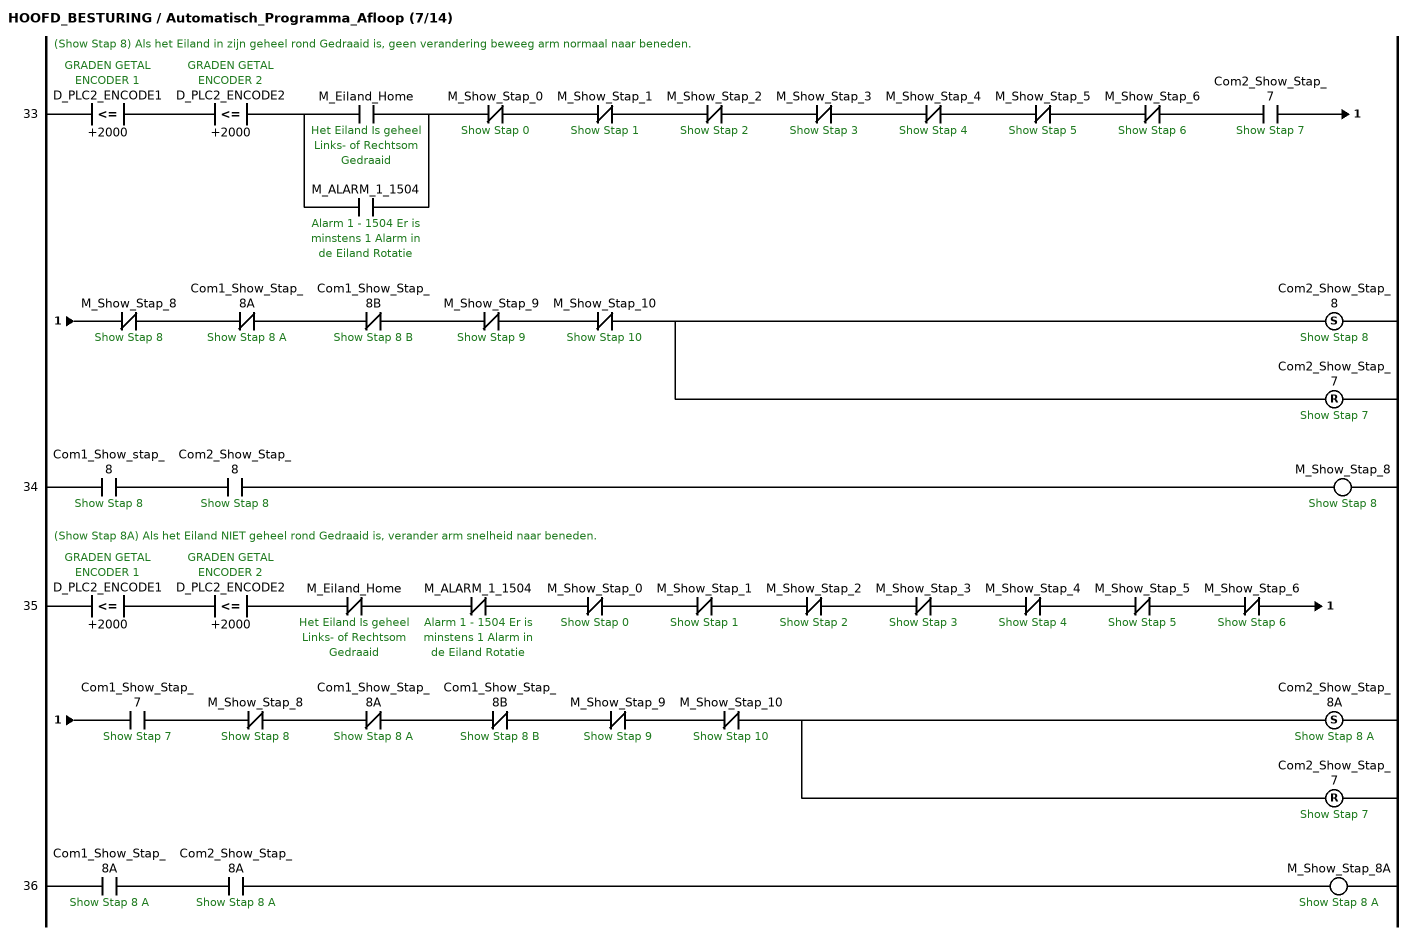
; rung 33: (Show Stap 8) Als het Eiland in zijn geheel rond Gedraaid is, geen verandering beweeg arm normaal naar beneden.
LD<=S(317) D_PLC2_ENCODE1 +2000  ; GRADEN GETAL ENCODER 1
AND<=S(317) D_PLC2_ENCODE2 +2000  ; GRADEN GETAL ENCODER 2
LD M_Eiland_Home  ; Het Eiland Is geheel Links- of Rechtsom Gedraaid
OR M_ALARM_1_1504  ; Alarm 1 - 1504 Er is minstens 1 Alarm in de Eiland Rotatie
ANDLD
ANDNOT M_Show_Stap_0  ; Show Stap 0
ANDNOT M_Show_Stap_1  ; Show Stap 1
ANDNOT M_Show_Stap_2  ; Show Stap 2
ANDNOT M_Show_Stap_3  ; Show Stap 3
ANDNOT M_Show_Stap_4  ; Show Stap 4
ANDNOT M_Show_Stap_5  ; Show Stap 5
ANDNOT M_Show_Stap_6  ; Show Stap 6
AND Com2_Show_Stap_7  ; Show Stap 7
ANDNOT M_Show_Stap_8  ; Show Stap 8
ANDNOT Com1_Show_Stap_8A  ; Show Stap 8 A
ANDNOT Com1_Show_Stap_8B  ; Show Stap 8 B
ANDNOT M_Show_Stap_9  ; Show Stap 9
ANDNOT M_Show_Stap_10  ; Show Stap 10
SET Com2_Show_Stap_8  ; Show Stap 8
RSET Com2_Show_Stap_7  ; Show Stap 7
; rung 34
LD Com1_Show_stap_8  ; Show Stap 8
AND Com2_Show_Stap_8  ; Show Stap 8
OUT M_Show_Stap_8  ; Show Stap 8
; rung 35: (Show Stap 8A) Als het Eiland NIET geheel rond Gedraaid is, verander arm snelheid naar beneden.
LD<=S(317) D_PLC2_ENCODE1 +2000  ; GRADEN GETAL ENCODER 1
AND<=S(317) D_PLC2_ENCODE2 +2000  ; GRADEN GETAL ENCODER 2
ANDNOT M_Eiland_Home  ; Het Eiland Is geheel Links- of Rechtsom Gedraaid
ANDNOT M_ALARM_1_1504  ; Alarm 1 - 1504 Er is minstens 1 Alarm in de Eiland Rotatie
ANDNOT M_Show_Stap_0  ; Show Stap 0
ANDNOT M_Show_Stap_1  ; Show Stap 1
ANDNOT M_Show_Stap_2  ; Show Stap 2
ANDNOT M_Show_Stap_3  ; Show Stap 3
ANDNOT M_Show_Stap_4  ; Show Stap 4
ANDNOT M_Show_Stap_5  ; Show Stap 5
ANDNOT M_Show_Stap_6  ; Show Stap 6
AND Com1_Show_Stap_7  ; Show Stap 7
ANDNOT M_Show_Stap_8  ; Show Stap 8
ANDNOT Com1_Show_Stap_8A  ; Show Stap 8 A
ANDNOT Com1_Show_Stap_8B  ; Show Stap 8 B
ANDNOT M_Show_Stap_9  ; Show Stap 9
ANDNOT M_Show_Stap_10  ; Show Stap 10
SET Com2_Show_Stap_8A  ; Show Stap 8 A
RSET Com2_Show_Stap_7  ; Show Stap 7
; rung 36
LD Com1_Show_Stap_8A  ; Show Stap 8 A
AND Com2_Show_Stap_8A  ; Show Stap 8 A
OUT M_Show_Stap_8A  ; Show Stap 8 A

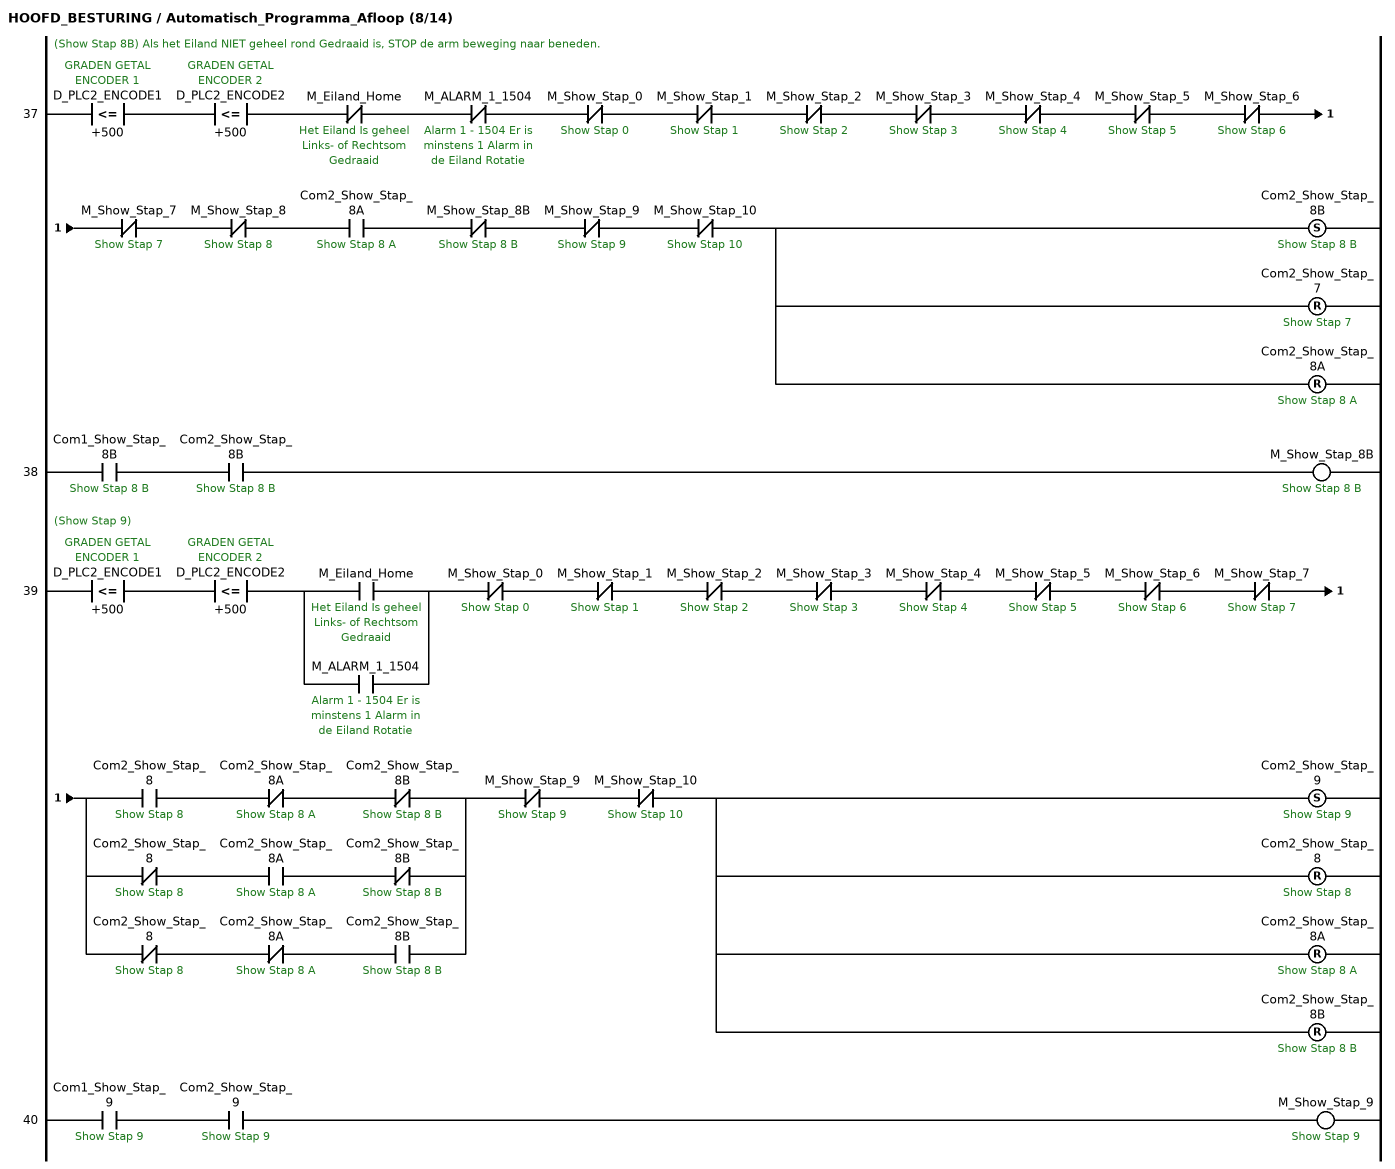
; rung 37: (Show Stap 8B) Als het Eiland NIET geheel rond Gedraaid is, STOP de arm beweging naar beneden.
LD<=S(317) D_PLC2_ENCODE1 +500  ; GRADEN GETAL ENCODER 1
AND<=S(317) D_PLC2_ENCODE2 +500  ; GRADEN GETAL ENCODER 2
ANDNOT M_Eiland_Home  ; Het Eiland Is geheel Links- of Rechtsom Gedraaid
ANDNOT M_ALARM_1_1504  ; Alarm 1 - 1504 Er is minstens 1 Alarm in de Eiland Rotatie
ANDNOT M_Show_Stap_0  ; Show Stap 0
ANDNOT M_Show_Stap_1  ; Show Stap 1
ANDNOT M_Show_Stap_2  ; Show Stap 2
ANDNOT M_Show_Stap_3  ; Show Stap 3
ANDNOT M_Show_Stap_4  ; Show Stap 4
ANDNOT M_Show_Stap_5  ; Show Stap 5
ANDNOT M_Show_Stap_6  ; Show Stap 6
ANDNOT M_Show_Stap_7  ; Show Stap 7
ANDNOT M_Show_Stap_8  ; Show Stap 8
AND Com2_Show_Stap_8A  ; Show Stap 8 A
ANDNOT M_Show_Stap_8B  ; Show Stap 8 B
ANDNOT M_Show_Stap_9  ; Show Stap 9
ANDNOT M_Show_Stap_10  ; Show Stap 10
SET Com2_Show_Stap_8B  ; Show Stap 8 B
RSET Com2_Show_Stap_7  ; Show Stap 7
RSET Com2_Show_Stap_8A  ; Show Stap 8 A
; rung 38
LD Com1_Show_Stap_8B  ; Show Stap 8 B
AND Com2_Show_Stap_8B  ; Show Stap 8 B
OUT M_Show_Stap_8B  ; Show Stap 8 B
; rung 39: (Show Stap 9)
LD<=S(317) D_PLC2_ENCODE1 +500  ; GRADEN GETAL ENCODER 1
AND<=S(317) D_PLC2_ENCODE2 +500  ; GRADEN GETAL ENCODER 2
LD M_Eiland_Home  ; Het Eiland Is geheel Links- of Rechtsom Gedraaid
OR M_ALARM_1_1504  ; Alarm 1 - 1504 Er is minstens 1 Alarm in de Eiland Rotatie
ANDLD
ANDNOT M_Show_Stap_0  ; Show Stap 0
ANDNOT M_Show_Stap_1  ; Show Stap 1
ANDNOT M_Show_Stap_2  ; Show Stap 2
ANDNOT M_Show_Stap_3  ; Show Stap 3
ANDNOT M_Show_Stap_4  ; Show Stap 4
ANDNOT M_Show_Stap_5  ; Show Stap 5
ANDNOT M_Show_Stap_6  ; Show Stap 6
ANDNOT M_Show_Stap_7  ; Show Stap 7
LD Com2_Show_Stap_8  ; Show Stap 8
ANDNOT Com2_Show_Stap_8A  ; Show Stap 8 A
ANDNOT Com2_Show_Stap_8B  ; Show Stap 8 B
LDNOT Com2_Show_Stap_8  ; Show Stap 8
AND Com2_Show_Stap_8A  ; Show Stap 8 A
ANDNOT Com2_Show_Stap_8B  ; Show Stap 8 B
ORLD
LDNOT Com2_Show_Stap_8  ; Show Stap 8
ANDNOT Com2_Show_Stap_8A  ; Show Stap 8 A
AND Com2_Show_Stap_8B  ; Show Stap 8 B
ORLD
ANDLD
ANDNOT M_Show_Stap_9  ; Show Stap 9
ANDNOT M_Show_Stap_10  ; Show Stap 10
SET Com2_Show_Stap_9  ; Show Stap 9
RSET Com2_Show_Stap_8  ; Show Stap 8
RSET Com2_Show_Stap_8A  ; Show Stap 8 A
RSET Com2_Show_Stap_8B  ; Show Stap 8 B
; rung 40
LD Com1_Show_Stap_9  ; Show Stap 9
AND Com2_Show_Stap_9  ; Show Stap 9
OUT M_Show_Stap_9  ; Show Stap 9

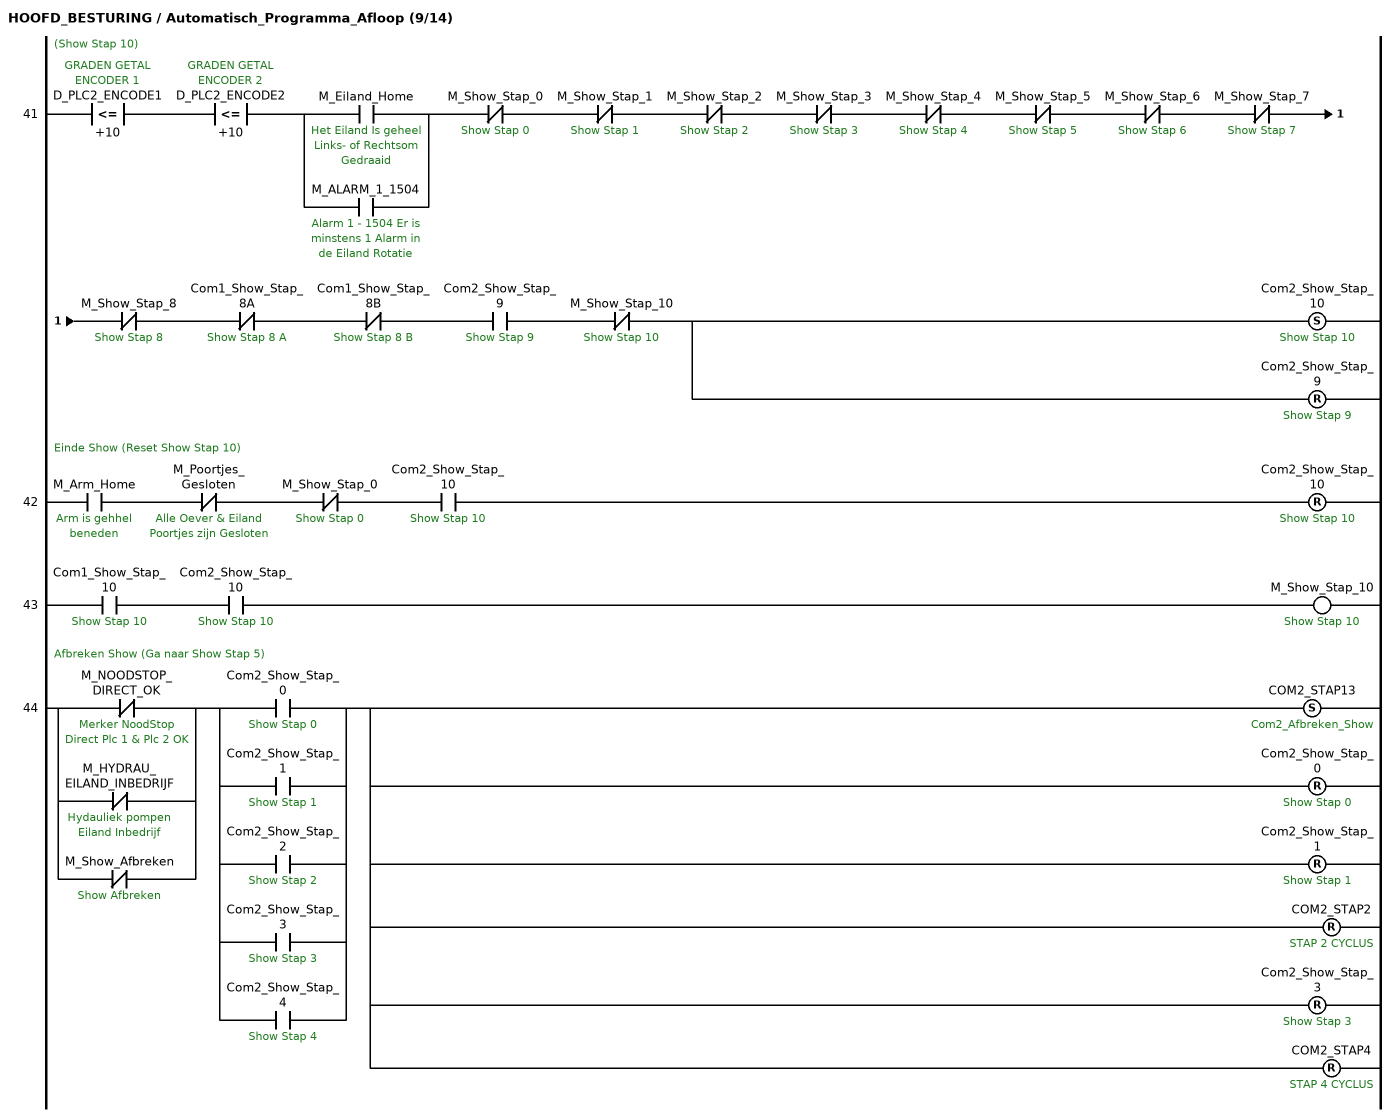
; rung 41: (Show Stap 10)
LD<=S(317) D_PLC2_ENCODE1 +10  ; GRADEN GETAL ENCODER 1
AND<=S(317) D_PLC2_ENCODE2 +10  ; GRADEN GETAL ENCODER 2
LD M_Eiland_Home  ; Het Eiland Is geheel Links- of Rechtsom Gedraaid
OR M_ALARM_1_1504  ; Alarm 1 - 1504 Er is minstens 1 Alarm in de Eiland Rotatie
ANDLD
ANDNOT M_Show_Stap_0  ; Show Stap 0
ANDNOT M_Show_Stap_1  ; Show Stap 1
ANDNOT M_Show_Stap_2  ; Show Stap 2
ANDNOT M_Show_Stap_3  ; Show Stap 3
ANDNOT M_Show_Stap_4  ; Show Stap 4
ANDNOT M_Show_Stap_5  ; Show Stap 5
ANDNOT M_Show_Stap_6  ; Show Stap 6
ANDNOT M_Show_Stap_7  ; Show Stap 7
ANDNOT M_Show_Stap_8  ; Show Stap 8
ANDNOT Com1_Show_Stap_8A  ; Show Stap 8 A
ANDNOT Com1_Show_Stap_8B  ; Show Stap 8 B
AND Com2_Show_Stap_9  ; Show Stap 9
ANDNOT M_Show_Stap_10  ; Show Stap 10
SET Com2_Show_Stap_10  ; Show Stap 10
RSET Com2_Show_Stap_9  ; Show Stap 9
; rung 42: Einde Show (Reset Show Stap 10)
LD M_Arm_Home  ; Arm is gehhel beneden
ANDNOT M_Poortjes_Gesloten  ; Alle Oever & Eiland Poortjes zijn Gesloten
ANDNOT M_Show_Stap_0  ; Show Stap 0
AND Com2_Show_Stap_10  ; Show Stap 10
RSET Com2_Show_Stap_10  ; Show Stap 10
; rung 43
LD Com1_Show_Stap_10  ; Show Stap 10
AND Com2_Show_Stap_10  ; Show Stap 10
OUT M_Show_Stap_10  ; Show Stap 10
; rung 44: Afbreken Show (Ga naar Show Stap 5)
LDNOT M_NOODSTOP_DIRECT_OK  ; Merker NoodStop Direct Plc 1 & Plc 2 OK
ORNOT M_HYDRAU_EILAND_INBEDRIJF  ; Hydauliek pompen Eiland Inbedrijf
ORNOT M_Show_Afbreken  ; Show Afbreken
LD Com2_Show_Stap_0  ; Show Stap 0
OR Com2_Show_Stap_1  ; Show Stap 1
OR Com2_Show_Stap_2  ; Show Stap 2
OR Com2_Show_Stap_3  ; Show Stap 3
OR Com2_Show_Stap_4  ; Show Stap 4
ANDLD
SET COM2_STAP13  ; Com2_Afbreken_Show
RSET Com2_Show_Stap_0  ; Show Stap 0
RSET Com2_Show_Stap_1  ; Show Stap 1
RSET COM2_STAP2  ; STAP 2 CYCLUS
RSET Com2_Show_Stap_3  ; Show Stap 3
RSET COM2_STAP4  ; STAP 4 CYCLUS

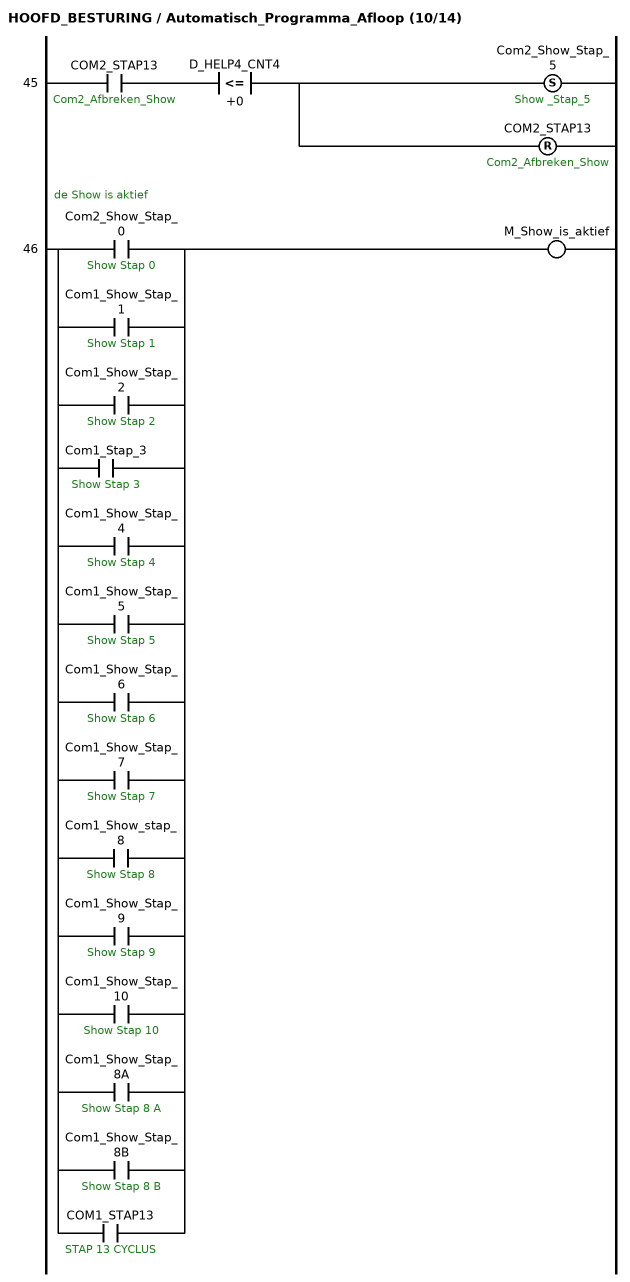
; rung 45
LD COM2_STAP13  ; Com2_Afbreken_Show
AND<=S(317) D_HELP4_CNT4 +0
SET Com2_Show_Stap_5  ; Show _Stap_5
RSET COM2_STAP13  ; Com2_Afbreken_Show
; rung 46: de Show is aktief
LD Com2_Show_Stap_0  ; Show Stap 0
OR Com1_Show_Stap_1  ; Show Stap 1
OR Com1_Show_Stap_2  ; Show Stap 2
OR Com1_Stap_3  ; Show Stap 3
OR Com1_Show_Stap_4  ; Show Stap 4
OR Com1_Show_Stap_5  ; Show Stap 5
OR Com1_Show_Stap_6  ; Show Stap 6
OR Com1_Show_Stap_7  ; Show Stap 7
OR Com1_Show_stap_8  ; Show Stap 8
OR Com1_Show_Stap_9  ; Show Stap 9
OR Com1_Show_Stap_10  ; Show Stap 10
OR Com1_Show_Stap_8A  ; Show Stap 8 A
OR Com1_Show_Stap_8B  ; Show Stap 8 B
OR COM1_STAP13  ; STAP 13 CYCLUS
OUT M_Show_is_aktief

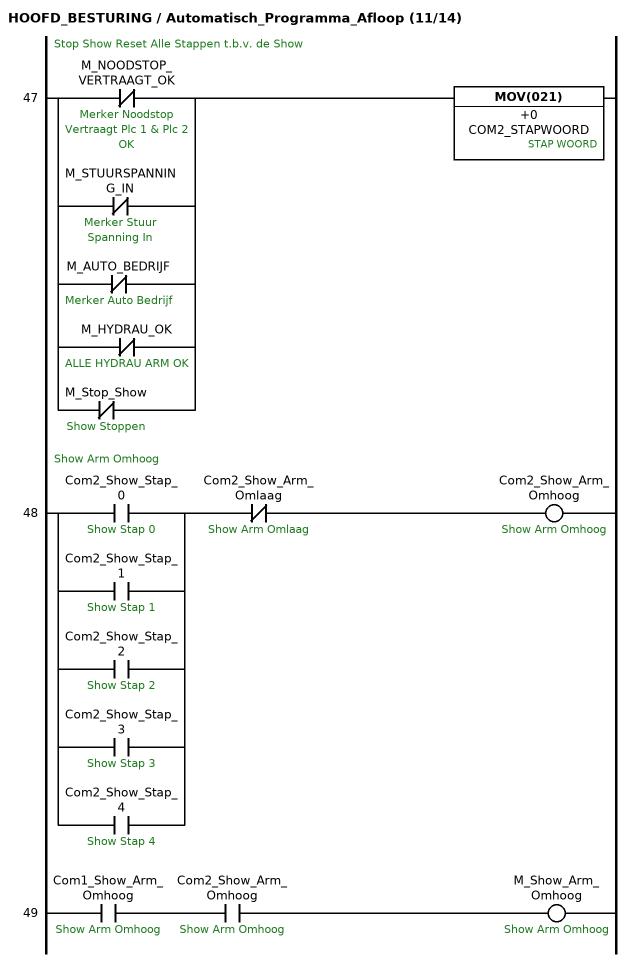
; rung 47: Stop Show Reset Alle Stappen t.b.v. de Show
LDNOT M_NOODSTOP_VERTRAAGT_OK  ; Merker Noodstop Vertraagt Plc 1 & Plc 2 OK
ORNOT M_STUURSPANNING_IN  ; Merker Stuur Spanning In
ORNOT M_AUTO_BEDRIJF  ; Merker Auto Bedrijf
ORNOT M_HYDRAU_OK  ; ALLE HYDRAU ARM OK
ORNOT M_Stop_Show  ; Show Stoppen
MOV(021) +0 COM2_STAPWOORD  ; STAP WOORD
; rung 48: Show Arm Omhoog
LD Com2_Show_Stap_0  ; Show Stap 0
OR Com2_Show_Stap_1  ; Show Stap 1
OR Com2_Show_Stap_2  ; Show Stap 2
OR Com2_Show_Stap_3  ; Show Stap 3
OR Com2_Show_Stap_4  ; Show Stap 4
ANDNOT Com2_Show_Arm_Omlaag  ; Show Arm Omlaag
OUT Com2_Show_Arm_Omhoog  ; Show Arm Omhoog
; rung 49
LD Com1_Show_Arm_Omhoog  ; Show Arm Omhoog
AND Com2_Show_Arm_Omhoog  ; Show Arm Omhoog
OUT M_Show_Arm_Omhoog  ; Show Arm Omhoog

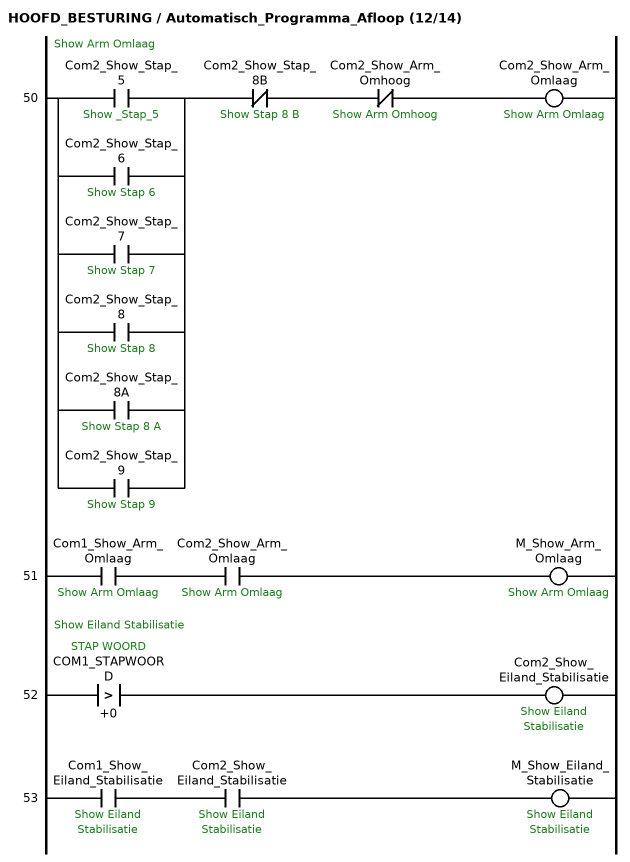
; rung 50: Show Arm Omlaag
LD Com2_Show_Stap_5  ; Show _Stap_5
OR Com2_Show_Stap_6  ; Show Stap 6
OR Com2_Show_Stap_7  ; Show Stap 7
OR Com2_Show_Stap_8  ; Show Stap 8
OR Com2_Show_Stap_8A  ; Show Stap 8 A
OR Com2_Show_Stap_9  ; Show Stap 9
ANDNOT Com2_Show_Stap_8B  ; Show Stap 8 B
ANDNOT Com2_Show_Arm_Omhoog  ; Show Arm Omhoog
OUT Com2_Show_Arm_Omlaag  ; Show Arm Omlaag
; rung 51
LD Com1_Show_Arm_Omlaag  ; Show Arm Omlaag
AND Com2_Show_Arm_Omlaag  ; Show Arm Omlaag
OUT M_Show_Arm_Omlaag  ; Show Arm Omlaag
; rung 52: Show Eiland Stabilisatie
LD>S(322) COM1_STAPWOORD +0  ; STAP WOORD
OUT Com2_Show_Eiland_Stabilisatie  ; Show Eiland Stabilisatie
; rung 53
LD Com1_Show_Eiland_Stabilisatie  ; Show Eiland Stabilisatie
AND Com2_Show_Eiland_Stabilisatie  ; Show Eiland Stabilisatie
OUT M_Show_Eiland_Stabilisatie  ; Show Eiland Stabilisatie

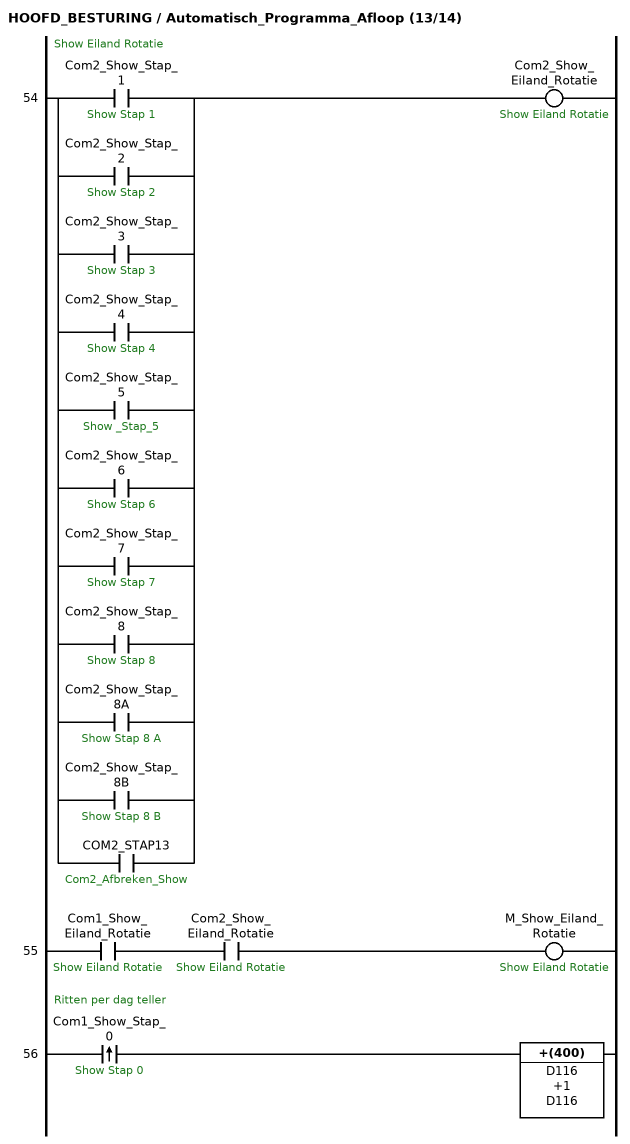
; rung 54: Show Eiland Rotatie
LD Com2_Show_Stap_1  ; Show Stap 1
OR Com2_Show_Stap_2  ; Show Stap 2
OR Com2_Show_Stap_3  ; Show Stap 3
OR Com2_Show_Stap_4  ; Show Stap 4
OR Com2_Show_Stap_5  ; Show _Stap_5
OR Com2_Show_Stap_6  ; Show Stap 6
OR Com2_Show_Stap_7  ; Show Stap 7
OR Com2_Show_Stap_8  ; Show Stap 8
OR Com2_Show_Stap_8A  ; Show Stap 8 A
OR Com2_Show_Stap_8B  ; Show Stap 8 B
OR COM2_STAP13  ; Com2_Afbreken_Show
OUT Com2_Show_Eiland_Rotatie  ; Show Eiland Rotatie
; rung 55
LD Com1_Show_Eiland_Rotatie  ; Show Eiland Rotatie
AND Com2_Show_Eiland_Rotatie  ; Show Eiland Rotatie
OUT M_Show_Eiland_Rotatie  ; Show Eiland Rotatie
; rung 56: Ritten per dag teller
@LD Com1_Show_Stap_0  ; Show Stap 0
+(400) D116 +1 D116

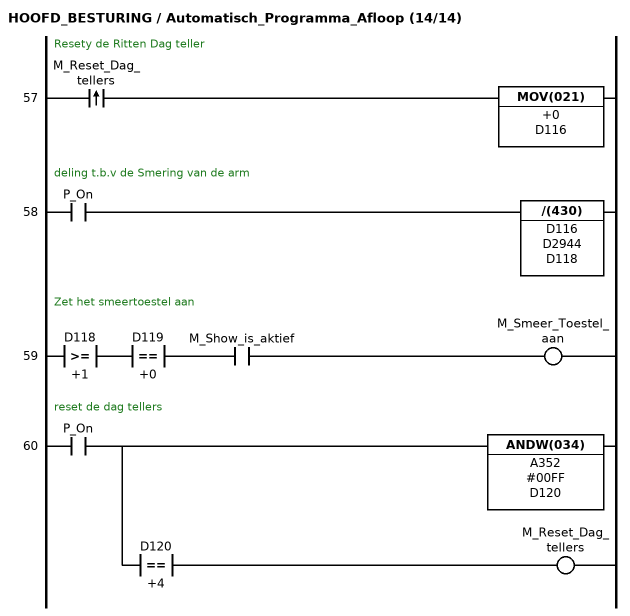
; rung 57: Resety de Ritten Dag teller
@LD M_Reset_Dag_tellers
MOV(021) +0 D116
; rung 58: deling t.b.v de Smering van de arm
LD P_On
/(430) D116 D2944 D118
; rung 59: Zet het smeertoestel aan
LD>=S(327) D118 +1
AND=S(302) D119 +0
AND M_Show_is_aktief
OUT M_Smeer_Toestel_aan
; rung 60: reset de dag tellers
LD P_On
ANDW(034) A352 #00FF D120
AND=S(302) D120 +4
OUT M_Reset_Dag_tellers

### Section Einde_Hoofd_Besturing
; rung 0
END(001)

## Program SIGNALEN_GROND (cyclic task 5)
Local symbols
D_ENCODE1_PLC2 UINT
D_ENC_1_PLUS_AFW D139 INT  ; ENCODER 1 + AFWIJKING
D_FACTOR_01 D5132 REAL  ; DIVERTION FACTOR IN REAL FORMAT
D_HELP2_CNT2 D5140 REAL  ; RESULT AFTER MULIPLYING IN REAL FORMAT
D_HELP3_CNT1 D5134 REAL  ; RESULT AFTER DIVERTING IN REAL FORMAT
D_HELP3_CNT2 D5144 REAL  ; RESULT AFTER DIVERTING IN REAL FORMAT

### Section Incremental_Encoder_Decoder_1

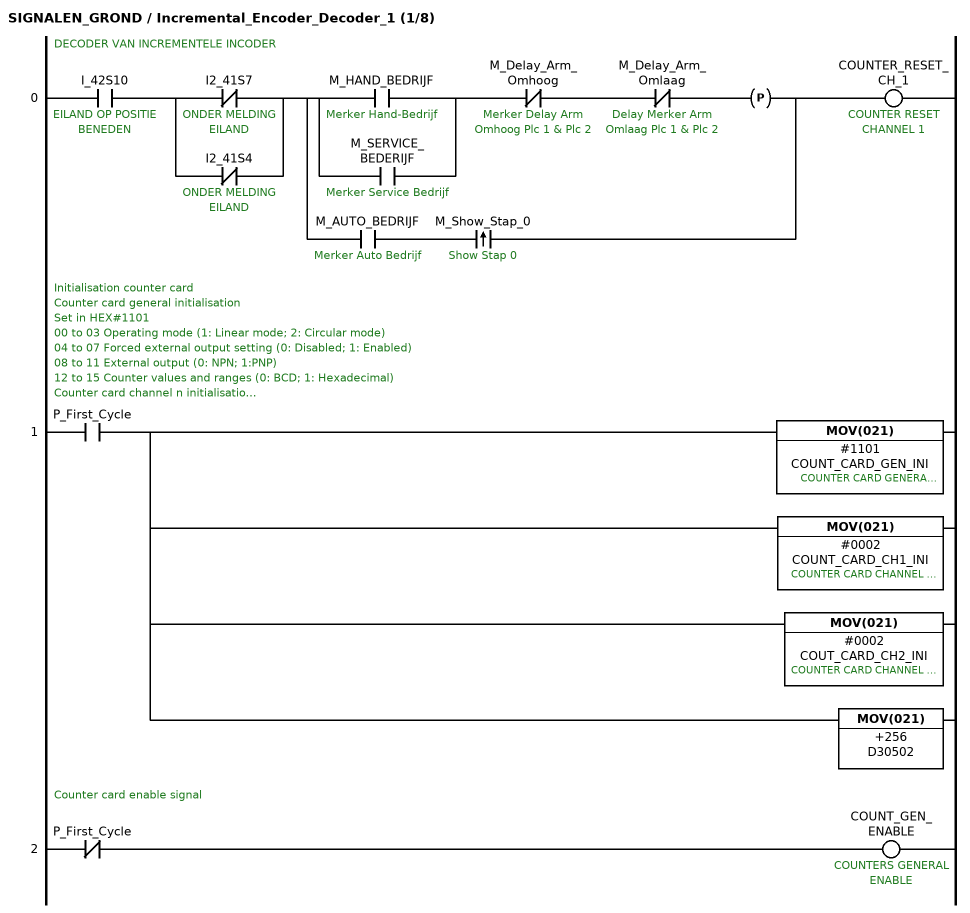
; rung 0: DECODER VAN INCREMENTELE INCODER
LD I_42S10  ; EILAND OP POSITIE BENEDEN
LDNOT I2_41S7  ; ONDER MELDING EILAND
ORNOT I2_41S4  ; ONDER MELDING EILAND
ANDLD
LD M_HAND_BEDRIJF  ; Merker Hand-Bedrijf
OR M_SERVICE_BEDERIJF  ; Merker Service Bedrijf
ANDNOT M_Delay_Arm_Omhoog  ; Merker Delay Arm Omhoog Plc 1 & Plc 2
ANDNOT M_Delay_Arm_Omlaag  ; Delay Merker Arm Omlaag Plc 1 & Plc 2
UP(521)
LD M_AUTO_BEDRIJF  ; Merker Auto Bedrijf
@AND M_Show_Stap_0  ; Show Stap 0
ORLD
ANDLD
OUT COUNTER_RESET_CH_1  ; COUNTER RESET CHANNEL 1
; rung 1: Initialisation counter card / Counter card general initialisation / Set in HEX#1101 / 00 to 03 Operating mode (1: Linear mode; 2: Circular mode) / 04 to 07 Forced external output setting (0: Disabled; 1: Enabled) / 08 to 11 External output (0: NPN; 1:PNP) / 12 to 15 Counter values and ranges (0: BCD; 1: Hexadecimal) / Counter card channel n initialisation / Set in HEX#0002 / 00 to 03 Counter 1 input types and counter reset conditions: / Input types / 0: x 1 / 1: x 2 / 2: x 4 / 3: Up and down pulses input / 4: Pulse and direction input / 04 to 07 Not used. / 08 to 15 Reset modes 00 to 11 (Mode 0 to mode 11)
LD P_First_Cycle
MOV(021) #1101 COUNT_CARD_GEN_INI  ; COUNTER CARD GENERAL INITIALISATION
MOV(021) #0002 COUNT_CARD_CH1_INI  ; COUNTER CARD CHANNEL 1 INITIALISATION
MOV(021) #0002 COUT_CARD_CH2_INI  ; COUNTER CARD CHANNEL 2 INITIALISATION
MOV(021) +256 D30502
; rung 2: Counter card enable signal
LDNOT P_First_Cycle
OUT COUNT_GEN_ENABLE  ; COUNTERS GENERAL ENABLE

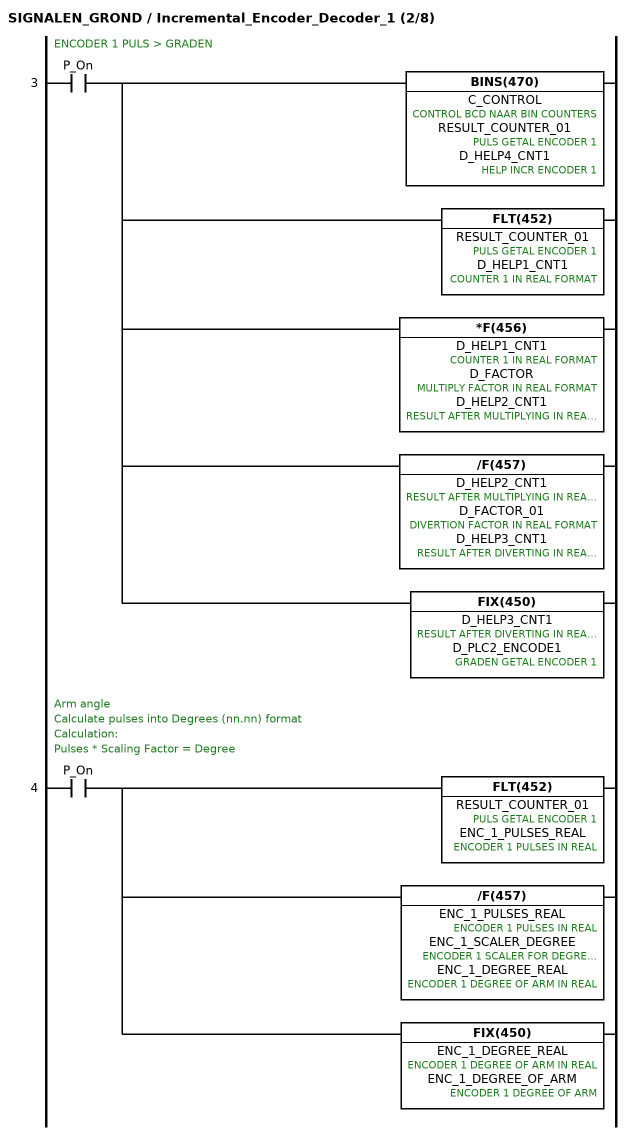
; rung 3: ENCODER 1 PULS > GRADEN
LD P_On
BINS(470) C_CONTROL RESULT_COUNTER_01 D_HELP4_CNT1  ; CONTROL BCD NAAR BIN COUNTERS, PULS GETAL ENCODER 1, HELP INCR ENCODER 1
FLT(452) RESULT_COUNTER_01 D_HELP1_CNT1  ; PULS GETAL ENCODER 1, COUNTER 1 IN REAL FORMAT
*F(456) D_HELP1_CNT1 D_FACTOR D_HELP2_CNT1  ; COUNTER 1 IN REAL FORMAT, MULTIPLY FACTOR IN REAL FORMAT, RESULT AFTER MULTIPLYING IN REAL FORMAT
/F(457) D_HELP2_CNT1 D_FACTOR_01 D_HELP3_CNT1  ; RESULT AFTER MULTIPLYING IN REAL FORMAT, DIVERTION FACTOR IN REAL FORMAT, RESULT AFTER DIVERTING IN REAL FORMAT
FIX(450) D_HELP3_CNT1 D_PLC2_ENCODE1  ; RESULT AFTER DIVERTING IN REAL FORMAT, GRADEN GETAL ENCODER 1
; rung 4: Arm angle / Calculate pulses into Degrees (nn.nn) format / Calculation: / Pulses * Scaling Factor = Degree
LD P_On
FLT(452) RESULT_COUNTER_01 ENC_1_PULSES_REAL  ; PULS GETAL ENCODER 1, ENCODER 1 PULSES IN REAL
/F(457) ENC_1_PULSES_REAL ENC_1_SCALER_DEGREE ENC_1_DEGREE_REAL  ; ENCODER 1 PULSES IN REAL, ENCODER 1 SCALER FOR DEGREE CALCULTION, ENCODER 1 DEGREE OF ARM IN REAL
FIX(450) ENC_1_DEGREE_REAL ENC_1_DEGREE_OF_ARM  ; ENCODER 1 DEGREE OF ARM IN REAL, ENCODER 1 DEGREE OF ARM

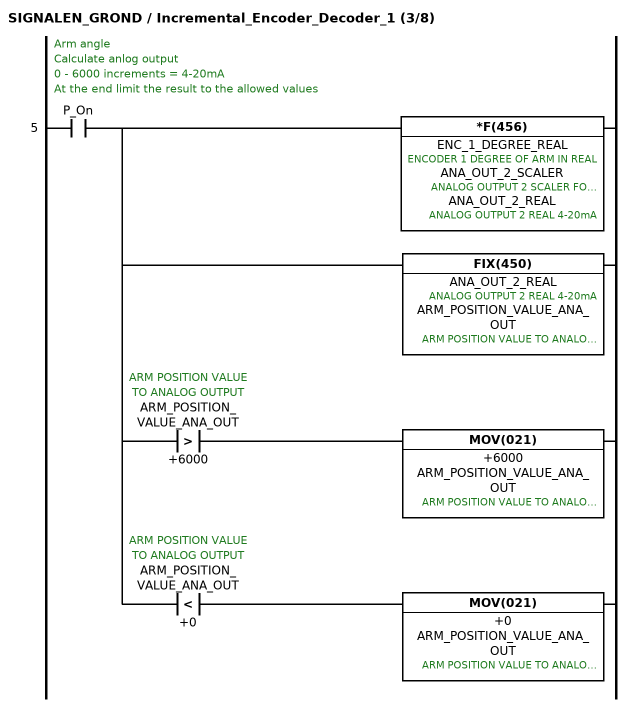
; rung 5: Arm angle / Calculate anlog output / 0 - 6000 increments = 4-20mA / At the end limit the result to the allowed values
LD P_On
OUT TR0
*F(456) ENC_1_DEGREE_REAL ANA_OUT_2_SCALER ANA_OUT_2_REAL  ; ENCODER 1 DEGREE OF ARM IN REAL, ANALOG OUTPUT 2 SCALER FOR 4-20mA, ANALOG OUTPUT 2 REAL 4-20mA
FIX(450) ANA_OUT_2_REAL ARM_POSITION_VALUE_ANA_OUT  ; ANALOG OUTPUT 2 REAL 4-20mA, ARM POSITION VALUE TO ANALOG OUTPUT
AND>S(322) ARM_POSITION_VALUE_ANA_OUT +6000  ; ARM POSITION VALUE TO ANALOG OUTPUT
MOV(021) +6000 ARM_POSITION_VALUE_ANA_OUT  ; ARM POSITION VALUE TO ANALOG OUTPUT
LD TR0
AND<S(312) ARM_POSITION_VALUE_ANA_OUT +0  ; ARM POSITION VALUE TO ANALOG OUTPUT
MOV(021) +0 ARM_POSITION_VALUE_ANA_OUT  ; ARM POSITION VALUE TO ANALOG OUTPUT

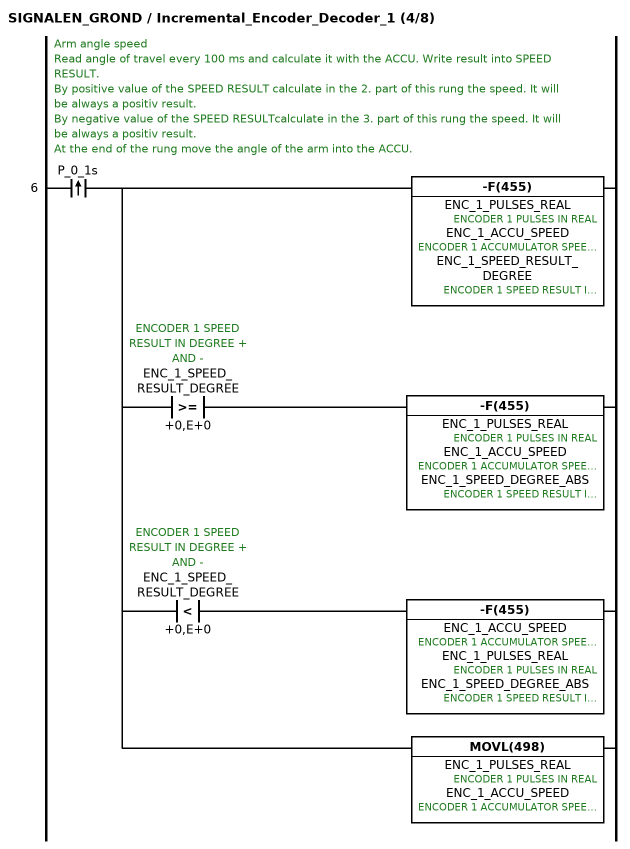
; rung 6: Arm angle speed / Read angle of travel every 100 ms and calculate it with the ACCU. Write result into SPEED RESULT. / By positive value of the SPEED RESULT calculate in the 2. part of this rung the speed. It will be always a positiv result. / By negative value of the SPEED RESULTcalculate in the 3. part of this rung the speed. It will be always a positiv result. / At the end of the rung move the angle of the arm into the ACCU.
@LD P_0_1s
OUT TR0
-F(455) ENC_1_PULSES_REAL ENC_1_ACCU_SPEED ENC_1_SPEED_RESULT_DEGREE  ; ENCODER 1 PULSES IN REAL, ENCODER 1 ACCUMULATOR SPEED CALCULATION, ENCODER 1 SPEED RESULT IN DEGREE + AND -
AND>=F(334) ENC_1_SPEED_RESULT_DEGREE +0,E+0  ; ENCODER 1 SPEED RESULT IN DEGREE + AND -
-F(455) ENC_1_PULSES_REAL ENC_1_ACCU_SPEED ENC_1_SPEED_DEGREE_ABS  ; ENCODER 1 PULSES IN REAL, ENCODER 1 ACCUMULATOR SPEED CALCULATION, ENCODER 1 SPEED RESULT IN DEGREE ABSOLUTE
LD TR0
AND<F(331) ENC_1_SPEED_RESULT_DEGREE +0,E+0  ; ENCODER 1 SPEED RESULT IN DEGREE + AND -
-F(455) ENC_1_ACCU_SPEED ENC_1_PULSES_REAL ENC_1_SPEED_DEGREE_ABS  ; ENCODER 1 ACCUMULATOR SPEED CALCULATION, ENCODER 1 PULSES IN REAL, ENCODER 1 SPEED RESULT IN DEGREE ABSOLUTE
LD TR0
MOVL(498) ENC_1_PULSES_REAL ENC_1_ACCU_SPEED  ; ENCODER 1 PULSES IN REAL, ENCODER 1 ACCUMULATOR SPEED CALCULATION

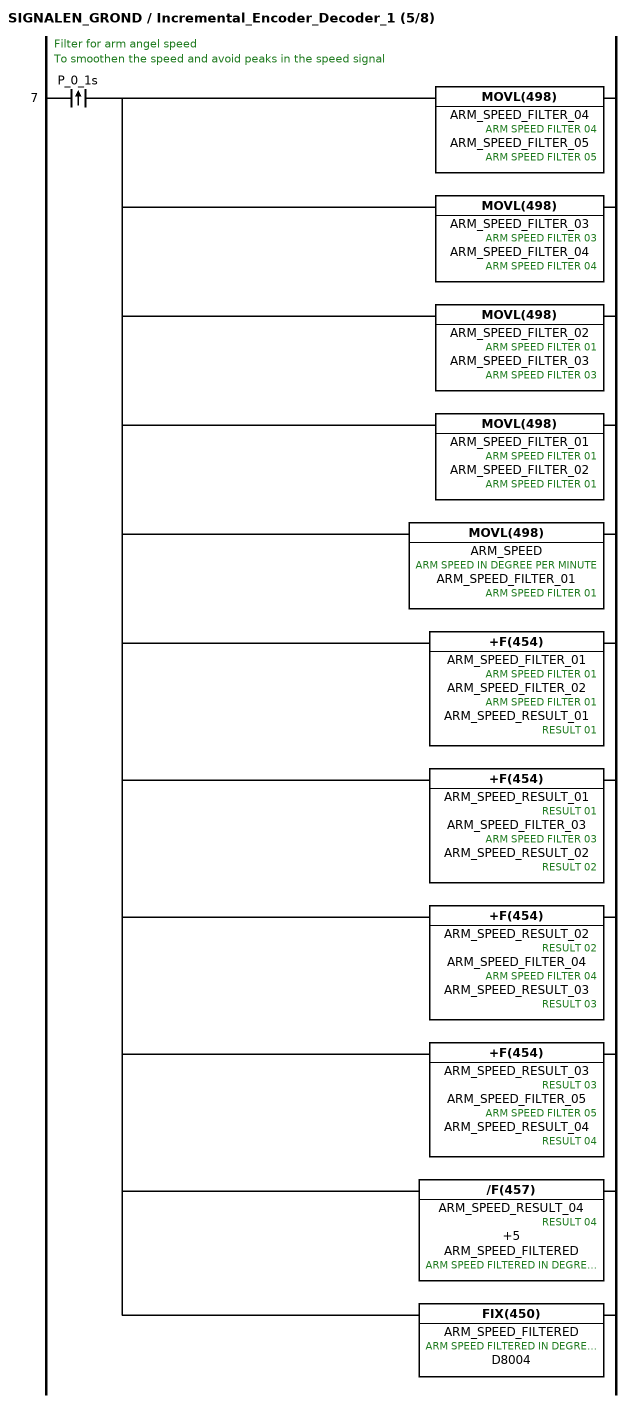
; rung 7: Filter for arm angel speed / To smoothen the speed and avoid peaks in the speed signal
@LD P_0_1s
MOVL(498) ARM_SPEED_FILTER_04 ARM_SPEED_FILTER_05  ; ARM SPEED FILTER 04, ARM SPEED FILTER 05
MOVL(498) ARM_SPEED_FILTER_03 ARM_SPEED_FILTER_04  ; ARM SPEED FILTER 03, ARM SPEED FILTER 04
MOVL(498) ARM_SPEED_FILTER_02 ARM_SPEED_FILTER_03  ; ARM SPEED FILTER 01, ARM SPEED FILTER 03
MOVL(498) ARM_SPEED_FILTER_01 ARM_SPEED_FILTER_02  ; ARM SPEED FILTER 01
MOVL(498) ARM_SPEED ARM_SPEED_FILTER_01  ; ARM SPEED IN DEGREE PER MINUTE, ARM SPEED FILTER 01
+F(454) ARM_SPEED_FILTER_01 ARM_SPEED_FILTER_02 ARM_SPEED_RESULT_01  ; ARM SPEED FILTER 01, RESULT 01
+F(454) ARM_SPEED_RESULT_01 ARM_SPEED_FILTER_03 ARM_SPEED_RESULT_02  ; RESULT 01, ARM SPEED FILTER 03, RESULT 02
+F(454) ARM_SPEED_RESULT_02 ARM_SPEED_FILTER_04 ARM_SPEED_RESULT_03  ; RESULT 02, ARM SPEED FILTER 04, RESULT 03
+F(454) ARM_SPEED_RESULT_03 ARM_SPEED_FILTER_05 ARM_SPEED_RESULT_04  ; RESULT 03, ARM SPEED FILTER 05, RESULT 04
/F(457) ARM_SPEED_RESULT_04 +5 ARM_SPEED_FILTERED  ; RESULT 04, ARM SPEED FILTERED IN DEGREE PER MINUTE
FIX(450) ARM_SPEED_FILTERED D8004  ; ARM SPEED FILTERED IN DEGREE PER MINUTE

